// TIA Portal V15.1 export
// export: Created 2024-05-17T05:38:48.6670872Z, ExportSetting WithDefaults, DisplayName Totally Integrated Automation Portal, DisplayVersion V15.1 Update 5, DisplayName TIA Portal Openness, DisplayVersion V15.1 Update 5, DisplayName SINAMICS Startdrive Advanced, DisplayVersion V15.1, DisplayName G130, G150, S120, S150, SINAMICS MV, S210, DisplayVersion V15.1, DisplayName G110M, G120, G120C, G120D, G120P, DisplayVersion V15.1, DisplayName STEP 7 Professional, DisplayVersion V15.1 Update 5, DisplayName STEP 7 Safety, DisplayVersion V15.1, DisplayName WinCC Professional, DisplayVersion V15.1 Update 5, DisplayName SIMATIC Visualization Architect, DisplayVersion V15.1
FUNCTION_BLOCK "LGBLiftTable3Pos1S4Det-MoviFitFCPN"   // FB6652, FBD
TITLE = LGBLiftTable3Pos1S4Det-MoviFitFCPN
{ S7_Optimized_Access := 'TRUE' }
AUTHOR : VCC
FAMILY : Tooling
VERSION : 0.0.0.0
// =============================================================================
// This module will be used for a unit with 2 stop positions, 1 speed and controlled by a
// SEW MoviFit PN frequency converter.
// It will get commands from higher level, evaluate the status of the interlock
// and give a finished in return when the task is completed.
// ============================================================================
// stored: AutoNumber false, IsIECCheckEnabled false, IsRetainMemResEnabled false, MemoryReserve 100, SetENOAutomatically False, UDAEnableTagReadback false
   VAR_INPUT
      I_PosSet { ExternalAccessible := 'False'; ExternalVisible := 'False'; ExternalWritable := 'False'} : Bool;   // Position Set Detection 1
      I_PosSetCheck { ExternalAccessible := 'False'; ExternalVisible := 'False'; ExternalWritable := 'False'} : Bool;   // Position Set Detection 2
      I_PosMiddle { ExternalAccessible := 'False'; ExternalVisible := 'False'; ExternalWritable := 'False'} : Bool;   // Position Middle Detection
      I_PosRes { ExternalAccessible := 'False'; ExternalVisible := 'False'; ExternalWritable := 'False'} : Bool;   // Position Reset Detection 1
      I_PosResCheck { ExternalAccessible := 'False'; ExternalVisible := 'False'; ExternalWritable := 'False'} : Bool;   // Position Reset Detection 2
      I_SetBegin { ExternalAccessible := 'False'; ExternalVisible := 'False'; ExternalWritable := 'False'} : Bool;   // Function Set begin selection
      I_MiddleBegin { ExternalAccessible := 'False'; ExternalVisible := 'False'; ExternalWritable := 'False'} : Bool;   // Function Middle begin selection
      I_ResBegin { ExternalAccessible := 'False'; ExternalVisible := 'False'; ExternalWritable := 'False'} : Bool;   // Function Reset begin selection
      I_PBSet { ExternalAccessible := 'False'; ExternalVisible := 'False'; ExternalWritable := 'False'} : Bool;   // Push button for Set direction used in manual
      I_PBReset { ExternalAccessible := 'False'; ExternalVisible := 'False'; ExternalWritable := 'False'} : Bool;   // Push button for reset direcion used in manual
      I_SetIntlkOK { ExternalAccessible := 'False'; ExternalVisible := 'False'; ExternalWritable := 'False'} : Bool;   // Set Interlock
      I_ResIntlkOK { ExternalAccessible := 'False'; ExternalVisible := 'False'; ExternalWritable := 'False'} : Bool;   // Reset Interlock
      I_MotorProtection { ExternalAccessible := 'False'; ExternalVisible := 'False'; ExternalWritable := 'False'} : Bool;   // Motor protection
      I_ReleaseBrake { ExternalAccessible := 'False'; ExternalVisible := 'False'; ExternalWritable := 'False'} : Bool;   // Release brake
      I_SafetyOk { ExternalAccessible := 'False'; ExternalVisible := 'False'; ExternalWritable := 'False'} : Bool;   // Safety Ok
      I_MotionStopOk { ExternalAccessible := 'False'; ExternalVisible := 'False'; ExternalWritable := 'False'} : Bool;   // Safety Ok / The motion stop is Ok
      I_HighSpeed { ExternalAccessible := 'False'; ExternalVisible := 'False'; ExternalWritable := 'False'} : Real;   // High speed Value (set-up %)
      I_SafetyStatusWord { ExternalAccessible := 'False'; ExternalVisible := 'False'; ExternalWritable := 'False'} : Word;   // Safety Status
      I_SafetyControlWord { ExternalAccessible := 'False'; ExternalVisible := 'False'; ExternalWritable := 'False'} : Word;   // Safety Control Word
   END_VAR
   VAR_OUTPUT
      O_SetPos { ExternalAccessible := 'False'; ExternalVisible := 'False'; ExternalWritable := 'False'} : Bool;   // In Position Set
      O_MiddlePos { ExternalAccessible := 'False'; ExternalVisible := 'False'; ExternalWritable := 'False'} : Bool;   // In Position Middle
      O_ResPos { ExternalAccessible := 'False'; ExternalVisible := 'False'; ExternalWritable := 'False'} : Bool;   // In Position Reset
      O_ReleaseBrake { ExternalAccessible := 'False'; ExternalVisible := 'False'; ExternalWritable := 'False'} : Bool;   // Release the brake of the motor
      O_Active { ExternalAccessible := 'False'; ExternalVisible := 'False'; ExternalWritable := 'False'} : Bool;   // Motor Active
      O_FuncRunning { ExternalAccessible := 'False'; ExternalVisible := 'False'; ExternalWritable := 'False'} : Bool;   // Signal that the function is busy
      O_SetFinished { ExternalAccessible := 'False'; ExternalVisible := 'False'; ExternalWritable := 'False'} : Bool;   // Function Set finished to Master Sequencing
      O_MiddleFinished { ExternalAccessible := 'False'; ExternalVisible := 'False'; ExternalWritable := 'False'} : Bool;   // Function Middle finished to Master Sequencing
      O_ResFinished { ExternalAccessible := 'False'; ExternalVisible := 'False'; ExternalWritable := 'False'} : Bool;   // Function Reset finished to Master Sequencing
      O_LEDSet { ExternalAccessible := 'False'; ExternalVisible := 'False'; ExternalWritable := 'False'} : Bool;   // Ledindication / Led indication for Set
      O_LEDMiddle { ExternalAccessible := 'False'; ExternalVisible := 'False'; ExternalWritable := 'False'} : Bool;   // Ledindication / Led indication for Middle
      O_LEDRes { ExternalAccessible := 'False'; ExternalVisible := 'False'; ExternalWritable := 'False'} : Bool;   // Ledindication / Led indication for Reset
      O_ReadyForOperation { ExternalAccessible := 'False'; ExternalVisible := 'False'; ExternalWritable := 'False'} : Bool;   // Ready for operation
      O_AlarmABCondition { ExternalAccessible := 'False'; ExternalVisible := 'False'; ExternalWritable := 'False'} : Bool;   // Alarm AB condition
      O_AlarmA { ExternalAccessible := 'False'; ExternalVisible := 'False'; ExternalWritable := 'False'} : Bool;   // Alarm A
      O_AlarmB { ExternalAccessible := 'False'; ExternalVisible := 'False'; ExternalWritable := 'False'} : Bool;   // Alarm B
      O_AlarmC { ExternalAccessible := 'False'; ExternalVisible := 'False'; ExternalWritable := 'False'} : Bool;   // Alarm C
      O_AlarmD { ExternalAccessible := 'False'; ExternalVisible := 'False'; ExternalWritable := 'False'} : Bool;   // Alarm D
      H_AlarmDWord { ExternalAccessible := 'False'; ExternalVisible := 'False'; ExternalWritable := 'False'} : DWord;   // Alarm Word
      H_AlarmDWord2 { ExternalAccessible := 'False'; ExternalVisible := 'False'; ExternalWritable := 'False'} : DWord;   // Alarm Word
   END_VAR
   VAR_IN_OUT
      IO_Modes : "Modes";
      C_Config : "LiftTable3Pos1S4DetMoviFitFCPNConfig";
      H_HMI : "H_HMI";
      "H_GBLiftTable3Pos1S4Det-MoviFitFCPN" : "H_GBLiftTable3Pos1S4Det-MoviFitFCPN";
   END_VAR
   VAR
      _MovFunc3Pos { ExternalAccessible := 'False'; ExternalVisible := 'False'; ExternalWritable := 'False'} : "LMovFnc3Pos";   // FB
      _StopPos { ExternalAccessible := 'False'; ExternalVisible := 'False'; ExternalWritable := 'False'} : "L3StopPos";   // FB
      _Motor { ExternalAccessible := 'False'; ExternalVisible := 'False'; ExternalWritable := 'False'} : "LGBMotor2W2S-MoviFitFCPN";   // FB
      _SetDetMissing { ExternalAccessible := 'False'; ExternalVisible := 'False'; ExternalWritable := 'False'} : "LTimer";   // Timer
      _ResDetMissing { ExternalAccessible := 'False'; ExternalVisible := 'False'; ExternalWritable := 'False'} : "LTimer";   // Timer
      H_FncSelInHMI { ExternalAccessible := 'False'; ExternalVisible := 'False'; ExternalWritable := 'False'} : Bool;
      AA_MotorProtection { ExternalAccessible := 'False'; ExternalVisible := 'False'; ExternalWritable := 'False'} : Bool;   // Motorprotection Not Ok / Motor Protection Tripped
      AA_SafetySwitch { ExternalAccessible := 'False'; ExternalVisible := 'False'; ExternalWritable := 'False'} : Bool;   // Safety Switch Not Ok
      AB_STO { ExternalAccessible := 'False'; ExternalVisible := 'False'; ExternalWritable := 'False'} : Bool;   // Safety Switch Not Ok / Safety output to drive is active but no response from drive that the safety is ok
      AB_Alarm { ExternalAccessible := 'False'; ExternalVisible := 'False'; ExternalWritable := 'False'} : Bool;   // Frequency Control / Alarm Frequency Control
      AB_KeepPosSetAlm { ExternalAccessible := 'False'; ExternalVisible := 'False'; ExternalWritable := 'False'} : Bool;   // Position Supervision Set Position / Lost Set Position
      AB_KeepPosMiddleAlm { ExternalAccessible := 'False'; ExternalVisible := 'False'; ExternalWritable := 'False'} : Bool;   // Position Supervision Set Position / Lost Middle Position
      AB_KeepPosResAlm { ExternalAccessible := 'False'; ExternalVisible := 'False'; ExternalWritable := 'False'} : Bool;   // Position Supervision Reset Position / Lost Reset Position
      AB_OvtSetAlm { ExternalAccessible := 'False'; ExternalVisible := 'False'; ExternalWritable := 'False'} : Bool;   // Timeout Set / TimeOut Set Direction
      AB_OvtMiddleAlm { ExternalAccessible := 'False'; ExternalVisible := 'False'; ExternalWritable := 'False'} : Bool;   // Timeout Set / TimeOut Middle Direction
      AB_OvtResAlm { ExternalAccessible := 'False'; ExternalVisible := 'False'; ExternalWritable := 'False'} : Bool;   // Timeout Reset / TimeOut Reset Direction
      AB_MoreDetAlm { ExternalAccessible := 'False'; ExternalVisible := 'False'; ExternalWritable := 'False'} : Bool;   // More than One Detection On at the same Time
      AB_SetDet1Missing { ExternalAccessible := 'False'; ExternalVisible := 'False'; ExternalWritable := 'False'} : Bool;   // Set Detector Signal Missing
      AB_SetDet2Missing { ExternalAccessible := 'False'; ExternalVisible := 'False'; ExternalWritable := 'False'} : Bool;   // Set Check Detector Signal Missing
      AB_ResDet1Missing { ExternalAccessible := 'False'; ExternalVisible := 'False'; ExternalWritable := 'False'} : Bool;   // Reset Detector Signal Missing
      AB_ResDet2Missing { ExternalAccessible := 'False'; ExternalVisible := 'False'; ExternalWritable := 'False'} : Bool;   // Reset Check Detector Signal Missing
      AC_KeepPosSetAlm { ExternalAccessible := 'False'; ExternalVisible := 'False'; ExternalWritable := 'False'} : Bool;   // Lost Set Position
      AC_KeepPosMiddleAlm { ExternalAccessible := 'False'; ExternalVisible := 'False'; ExternalWritable := 'False'} : Bool;   // Lost Set Position / Lost Middle Position
      AC_KeepPosResAlm { ExternalAccessible := 'False'; ExternalVisible := 'False'; ExternalWritable := 'False'} : Bool;   // Lost Reset Position
      AC_OvtSetAlm { ExternalAccessible := 'False'; ExternalVisible := 'False'; ExternalWritable := 'False'} : Bool;   // Timeout Set / TimeOut Set Direction
      AC_OvtMiddleAlm { ExternalAccessible := 'False'; ExternalVisible := 'False'; ExternalWritable := 'False'} : Bool;   // Timeout Set / TimeOut Middle Direction
      AC_OvtResAlm { ExternalAccessible := 'False'; ExternalVisible := 'False'; ExternalWritable := 'False'} : Bool;   // Timeout Reset / TimeOut Reset Direction
      AC_MoreDetAlm { ExternalAccessible := 'False'; ExternalVisible := 'False'; ExternalWritable := 'False'} : Bool;   // More than One Detection On at the same Time
      AC_SetDet1Missing { ExternalAccessible := 'False'; ExternalVisible := 'False'; ExternalWritable := 'False'} : Bool;   // Set Detector Signal Missing
      AC_SetDet2Missing { ExternalAccessible := 'False'; ExternalVisible := 'False'; ExternalWritable := 'False'} : Bool;   // Set Check Detector Signal Missing
      AC_ResDet1Missing { ExternalAccessible := 'False'; ExternalVisible := 'False'; ExternalWritable := 'False'} : Bool;   // Reset Detector Signal Missing
      AC_ResDet2Missing { ExternalAccessible := 'False'; ExternalVisible := 'False'; ExternalWritable := 'False'} : Bool;   // Reset Check Detector Signal Missing
      AD_OvtSetWarn { ExternalAccessible := 'False'; ExternalVisible := 'False'; ExternalWritable := 'False'} : Bool;   // Timeout Set / TimeOut Set Direction
      AD_OvtMiddleWarn { ExternalAccessible := 'False'; ExternalVisible := 'False'; ExternalWritable := 'False'} : Bool;   // TimeOut To Middle / Timeout Middle
      AD_OvtResWarn { ExternalAccessible := 'False'; ExternalVisible := 'False'; ExternalWritable := 'False'} : Bool;   // Timeout Reset / TimeOut Reset Direction
      AD_IntlkSetAlm { ExternalAccessible := 'False'; ExternalVisible := 'False'; ExternalWritable := 'False'} : Bool;   // Interlock Set
      AD_IntlkMiddleAlm { ExternalAccessible := 'False'; ExternalVisible := 'False'; ExternalWritable := 'False'} : Bool;   // Interlock Middle
      AD_IntlkResAlm { ExternalAccessible := 'False'; ExternalVisible := 'False'; ExternalWritable := 'False'} : Bool;   // Interlock Reset
      AD_Warning { ExternalAccessible := 'False'; ExternalVisible := 'False'; ExternalWritable := 'False'} : Bool;   // Frequency Control / Warning Frequency Control
      AA_NoBusControl { ExternalAccessible := 'False'; ExternalVisible := 'False'; ExternalWritable := 'False'} : Bool;   // Bus control inactive / Bus Control Inactive Frequency Control
      AD_MotionStop { ExternalAccessible := 'False'; ExternalVisible := 'False'; ExternalWritable := 'False'} : Bool;   // Motion Stop
      AC_ConfigCalibrationAlm { ExternalAccessible := 'False'; ExternalVisible := 'False'; ExternalWritable := 'False'} : Bool;   // The Config values for Warming/Alarm time must be ALL zero or ALL different from zero
      AD_CalibrationWarn { ExternalAccessible := 'False'; ExternalVisible := 'False'; ExternalWritable := 'False'} : Bool;   // No High speed selected so Calibration is not possible
      AC_ConfigRampAlm { ExternalAccessible := 'False'; ExternalVisible := 'False'; ExternalWritable := 'False'} : Bool;   // The config value for the ramp is not correct, must be zero or the config values for the calculation of the ramp must be ALL zero
      AC_ConfigRampCalcAlm { ExternalAccessible := 'False'; ExternalVisible := 'False'; ExternalWritable := 'False'} : Bool;   // The config values for the calculation of the ramp must be ALL different from zero
      PODataNotEnabled { ExternalAccessible := 'False'; ExternalVisible := 'False'; ExternalWritable := 'False'} : Bool;   // Bus control inactive
      SafetyOk { ExternalAccessible := 'False'; ExternalVisible := 'False'; ExternalWritable := 'False'} : Bool;   // Safety Ok
      SetPos { ExternalAccessible := 'False'; ExternalVisible := 'False'; ExternalWritable := 'False'} : Bool;   // Set position
      MiddlePos { ExternalAccessible := 'False'; ExternalVisible := 'False'; ExternalWritable := 'False'} : Bool;   // Middle Position
      ResPos { ExternalAccessible := 'False'; ExternalVisible := 'False'; ExternalWritable := 'False'} : Bool;   // Reset position
      AlarmA { ExternalAccessible := 'False'; ExternalVisible := 'False'; ExternalWritable := 'False'} : Bool;   // Alarm A
      AlarmB { ExternalAccessible := 'False'; ExternalVisible := 'False'; ExternalWritable := 'False'} : Bool;   // Alarm B
      AlarmC { ExternalAccessible := 'False'; ExternalVisible := 'False'; ExternalWritable := 'False'} : Bool;   // Alarm C
      AlarmD { ExternalAccessible := 'False'; ExternalVisible := 'False'; ExternalWritable := 'False'} : Bool;   // Alarm D
      SetIntlkOK { ExternalAccessible := 'False'; ExternalVisible := 'False'; ExternalWritable := 'False'} : Bool;   // Set Interlock
      MiddleIntlkOK { ExternalAccessible := 'False'; ExternalVisible := 'False'; ExternalWritable := 'False'} : Bool;   // Set Interlock / Middle Interlock
      ResIntlkOK { ExternalAccessible := 'False'; ExternalVisible := 'False'; ExternalWritable := 'False'} : Bool;   // Reset Interlock
      FuncRunning { ExternalAccessible := 'False'; ExternalVisible := 'False'; ExternalWritable := 'False'} : Bool;   // Function running
      MovFuncAlmCond { ExternalAccessible := 'False'; ExternalVisible := 'False'; ExternalWritable := 'False'} : Bool;   // Move function Alarm Condition
      StopPosAlmCond { ExternalAccessible := 'False'; ExternalVisible := 'False'; ExternalWritable := 'False'} : Bool;   // Stop posistion Alarm Condition
      KeepPosSetAlm { ExternalAccessible := 'False'; ExternalVisible := 'False'; ExternalWritable := 'False'} : Bool;   // Alarm Keep Position Set Position
      KeepPosMiddleAlm { ExternalAccessible := 'False'; ExternalVisible := 'False'; ExternalWritable := 'False'} : Bool;   // Keep Position Middle Alarm
      KeepPosResAlm { ExternalAccessible := 'False'; ExternalVisible := 'False'; ExternalWritable := 'False'} : Bool;   // Position Supervision Reset Position
      OvtSetAlm { ExternalAccessible := 'False'; ExternalVisible := 'False'; ExternalWritable := 'False'} : Bool;   // Timeout Set
      OvtMiddleAlm { ExternalAccessible := 'False'; ExternalVisible := 'False'; ExternalWritable := 'False'} : Bool;   // Overtime goto Middle Alarm
      OvtResAlm { ExternalAccessible := 'False'; ExternalVisible := 'False'; ExternalWritable := 'False'} : Bool;   // Overtime reset Alarm
      OneSetDetMissing { ExternalAccessible := 'False'; ExternalVisible := 'False'; ExternalWritable := 'False'} : Bool;   // One Set detector is missing
      OneResDetMissing { ExternalAccessible := 'False'; ExternalVisible := 'False'; ExternalWritable := 'False'} : Bool;   // One Reset detector is missing
      DetectorMissing { ExternalAccessible := 'False'; ExternalVisible := 'False'; ExternalWritable := 'False'} : Bool;   // One detector is missing
      OutOfUse { ExternalAccessible := 'False'; ExternalVisible := 'False'; ExternalWritable := 'False'} : Bool;   // Out of use
      MotorLoopAlarmCond { ExternalAccessible := 'False'; ExternalVisible := 'False'; ExternalWritable := 'False'} : Bool;   // Motor loop Alarm Condition
      ReadyForOperation { ExternalAccessible := 'False'; ExternalVisible := 'False'; ExternalWritable := 'False'} : Bool;   // Motor Loop Ready for operation
      MotorLoopActive { ExternalAccessible := 'False'; ExternalVisible := 'False'; ExternalWritable := 'False'} : Bool;   // Motor Loop Active
      AlarmABCondition { ExternalAccessible := 'False'; ExternalVisible := 'False'; ExternalWritable := 'False'} : Bool;   // Alarm AB Condition
      ReleaseBrake { ExternalAccessible := 'False'; ExternalVisible := 'False'; ExternalWritable := 'False'} : Bool;   // Release brake
      MotorCmdSet { ExternalAccessible := 'False'; ExternalVisible := 'False'; ExternalWritable := 'False'} : Bool;   // Command to motorloop set
      MotorCmdRes { ExternalAccessible := 'False'; ExternalVisible := 'False'; ExternalWritable := 'False'} : Bool;   // Command to motorloop reset
      SetPosDelayd { ExternalAccessible := 'False'; ExternalVisible := 'False'; ExternalWritable := 'False'} : Bool;   // Set Position Delayed
      MiddlePosDelayd { ExternalAccessible := 'False'; ExternalVisible := 'False'; ExternalWritable := 'False'} : Bool;   // Middle Position Delayed
      ResPosDelayd { ExternalAccessible := 'False'; ExternalVisible := 'False'; ExternalWritable := 'False'} : Bool;   // Reset Position Delayed
   END_VAR
   VAR RETAIN
      MemPrevPosRes { ExternalAccessible := 'False'; ExternalVisible := 'False'; ExternalWritable := 'False'} : Bool;   // Memory previous position was Reset
   END_VAR
   VAR
      MoreThenOneDetAlm { ExternalAccessible := 'False'; ExternalVisible := 'False'; ExternalWritable := 'False'} : Bool;   // More then one detection Alarm
      CmdSet { ExternalAccessible := 'False'; ExternalVisible := 'False'; ExternalWritable := 'False'} : Bool;   // Command Set
      CmdMiddle { ExternalAccessible := 'False'; ExternalVisible := 'False'; ExternalWritable := 'False'} : Bool;   // Command Middle
      CmdRes { ExternalAccessible := 'False'; ExternalVisible := 'False'; ExternalWritable := 'False'} : Bool;   // Command Reset
      MiddleStartMan { ExternalAccessible := 'False'; ExternalVisible := 'False'; ExternalWritable := 'False'} : Bool;   // Middle pos reached
      MiddleReachedMan { ExternalAccessible := 'False'; ExternalVisible := 'False'; ExternalWritable := 'False'} : Bool;   // Middle pos reached
      MiddleReachedManSTOP { ExternalAccessible := 'False'; ExternalVisible := 'False'; ExternalWritable := 'False'} : Bool;   // Middle pos reached
      PosSetDelayTimer { ExternalAccessible := 'False'; ExternalVisible := 'False'; ExternalWritable := 'False'} : "LTimer";   // FB
      PosMiddleDelayTimer { ExternalAccessible := 'False'; ExternalVisible := 'False'; ExternalWritable := 'False'} : "LTimer";   // FB
      PosResDelayTimer { ExternalAccessible := 'False'; ExternalVisible := 'False'; ExternalWritable := 'False'} : "LTimer";   // FB
   END_VAR
   VAR_TEMP
      H_HMITemp : "H_HMI";   // Animation
      H_HMIMotor : "H_HMI";   // Temp
      TempDInt : DInt;   // Temp DInt
      RunTimeMaxMiddleWarn : DInt;   // Time in ms for overtime warning
      RunTimeMaxMiddleAlm : DInt;   // Time in ms for overtime alarm
   END_VAR
   VAR_TEMP   // added for the SCL form of the ladder/FBD networks
      _w1 : Bool;
   END_VAR
BEGIN

REGION Network 1: **** 1 - Inputs **** Set Position Delay Timer
   // Set Position Delay Timer
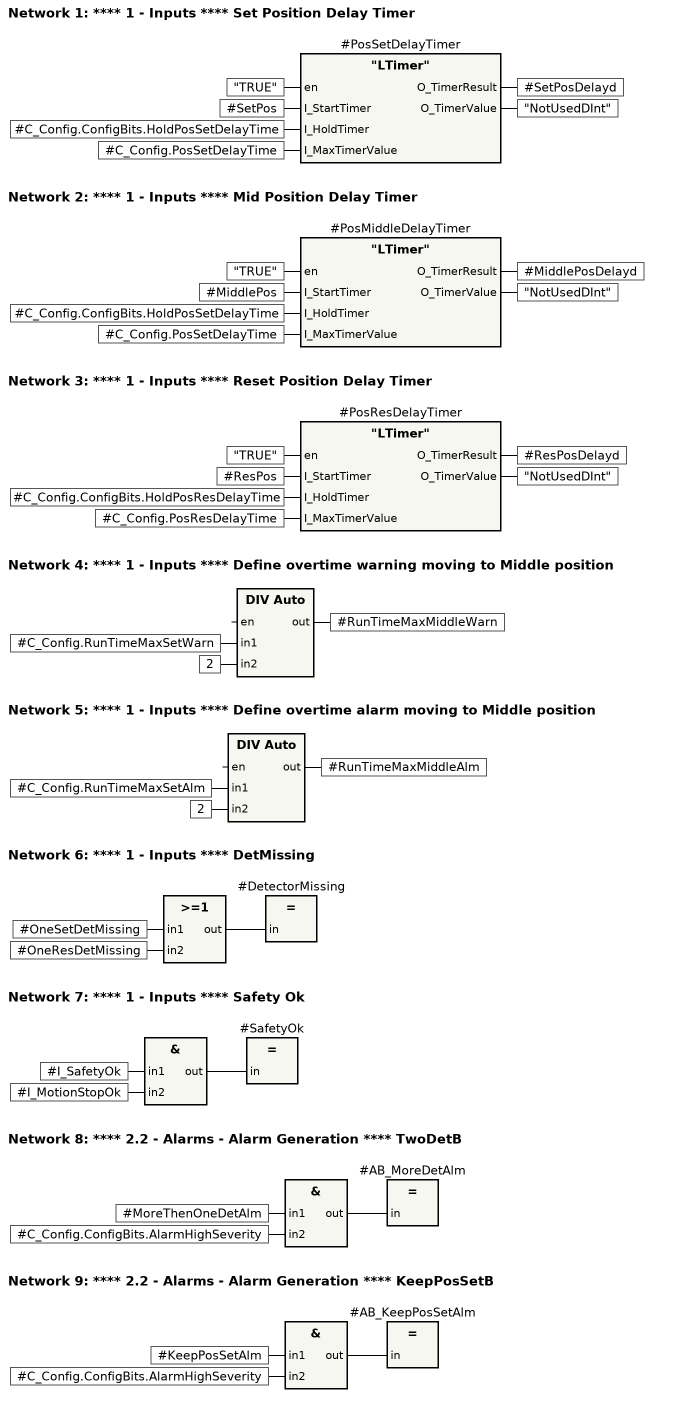
   IF "TRUE" THEN
       #PosSetDelayTimer(I_StartTimer := #SetPos,   // "LTimer"
                         I_HoldTimer := #C_Config.ConfigBits.HoldPosSetDelayTime,
                         I_MaxTimerValue := #C_Config.PosSetDelayTime,
                         O_TimerResult => #SetPosDelayd,
                         O_TimerValue => "NotUsedDInt");
   END_IF;
END_REGION

REGION Network 2: **** 1 - Inputs **** Mid Position Delay Timer
   // Middle Position Delay Timer
   IF "TRUE" THEN
       #PosMiddleDelayTimer(I_StartTimer := #MiddlePos,   // "LTimer"
                            I_HoldTimer := #C_Config.ConfigBits.HoldPosSetDelayTime,
                            I_MaxTimerValue := #C_Config.PosSetDelayTime,
                            O_TimerResult => #MiddlePosDelayd,
                            O_TimerValue => "NotUsedDInt");
   END_IF;
END_REGION

REGION Network 3: **** 1 - Inputs **** Reset Position Delay Timer
   // Reset Position Delay Timer
   IF "TRUE" THEN
       #PosResDelayTimer(I_StartTimer := #ResPos,   // "LTimer"
                         I_HoldTimer := #C_Config.ConfigBits.HoldPosResDelayTime,
                         I_MaxTimerValue := #C_Config.PosResDelayTime,
                         O_TimerResult => #ResPosDelayd,
                         O_TimerValue => "NotUsedDInt");
   END_IF;
END_REGION

REGION Network 4: **** 1 - Inputs **** Define overtime warning moving to Middle position
   // Define overtime warning moving to Middle position
   #RunTimeMaxMiddleWarn := #C_Config.RunTimeMaxSetWarn / 2;
END_REGION

REGION Network 5: **** 1 - Inputs **** Define overtime alarm moving to Middle position
   // Define overtime alarm moving to Middle position
   #RunTimeMaxMiddleAlm := #C_Config.RunTimeMaxSetAlm / 2;
END_REGION

REGION Network 6: **** 1 - Inputs **** DetMissing
   // Disable other Alarms when a detector is missing
   #DetectorMissing := #OneSetDetMissing OR #OneResDetMissing;
END_REGION

REGION Network 7: **** 1 - Inputs **** Safety Ok
   #SafetyOk := #I_SafetyOk AND #I_MotionStopOk;
END_REGION

REGION Network 8: **** 2.2 - Alarms - Alarm Generation **** TwoDetB
   // Two Detection B Alarm
   #AB_MoreDetAlm := #MoreThenOneDetAlm AND #C_Config.ConfigBits.AlarmHighSeverity;
END_REGION

REGION Network 9: **** 2.2 - Alarms - Alarm Generation **** KeepPosSetB
   // Keep position Set B Alarm
   #AB_KeepPosSetAlm := #KeepPosSetAlm AND #C_Config.ConfigBits.AlarmHighSeverity;
END_REGION

REGION Network 10: **** 2.2 - Alarms - Alarm Generation **** KeepPosSetB / **** 2.2 - Alarms - Alarm Generation **** KeepPosMiddleB
   // Keep position Set B Alarm / Keep position Middle B Alarm
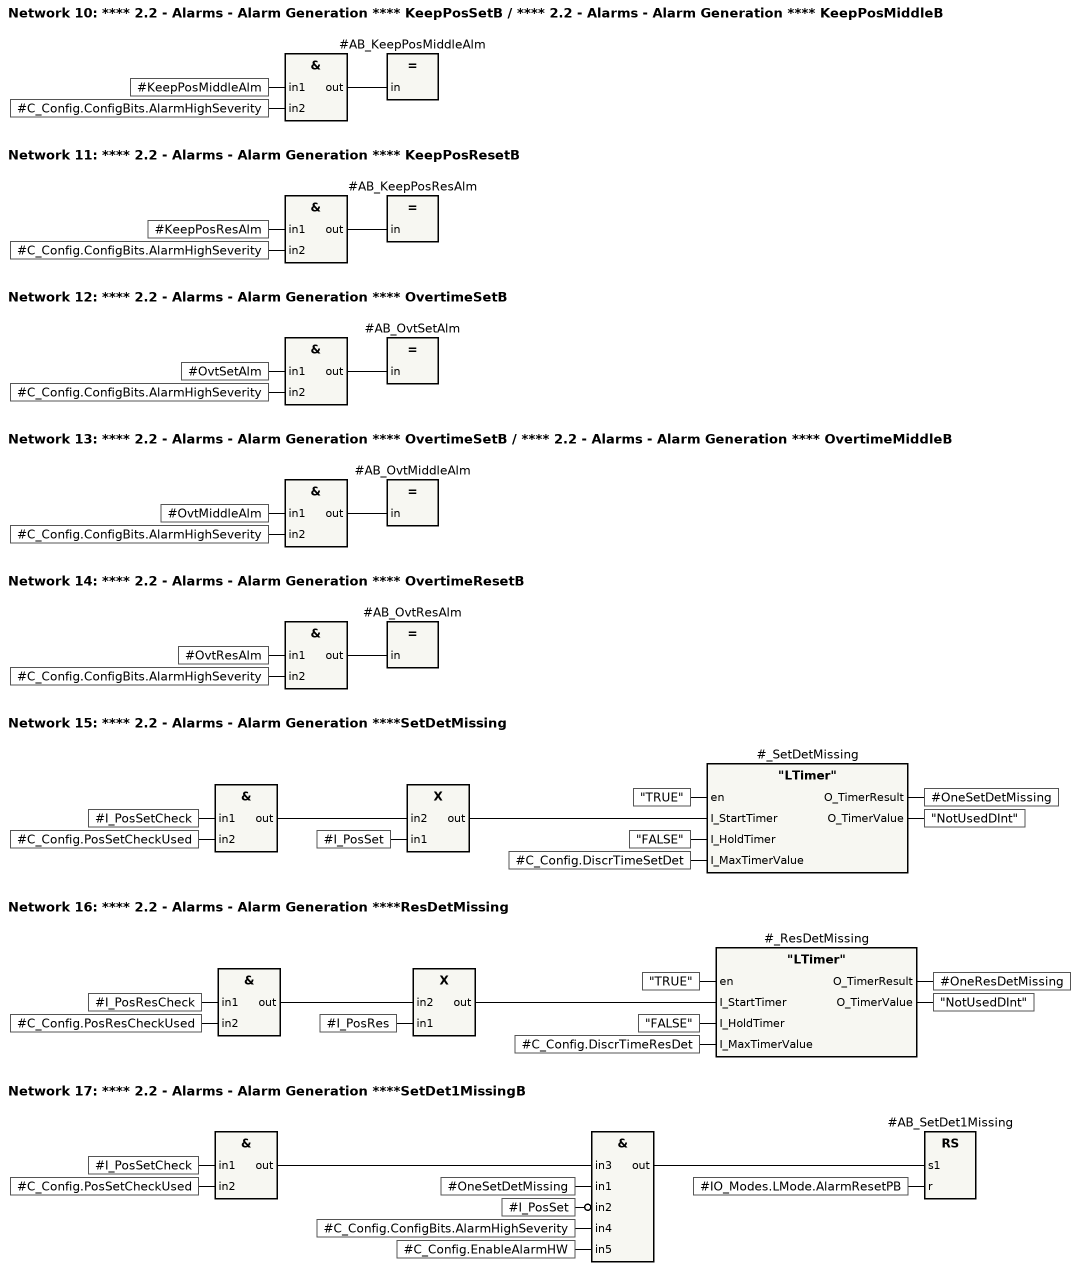
   #AB_KeepPosMiddleAlm := #KeepPosMiddleAlm AND #C_Config.ConfigBits.AlarmHighSeverity;
END_REGION

REGION Network 11: **** 2.2 - Alarms - Alarm Generation **** KeepPosResetB
   // Keep position reset B Alarm
   #AB_KeepPosResAlm := #KeepPosResAlm AND #C_Config.ConfigBits.AlarmHighSeverity;
END_REGION

REGION Network 12: **** 2.2 - Alarms - Alarm Generation **** OvertimeSetB
   // Overtime set B Alarm
   #AB_OvtSetAlm := #OvtSetAlm AND #C_Config.ConfigBits.AlarmHighSeverity;
END_REGION

REGION Network 13: **** 2.2 - Alarms - Alarm Generation **** OvertimeSetB / **** 2.2 - Alarms - Alarm Generation **** OvertimeMiddleB
   // Overtime set B Alarm / Overtime Middle B Alarm
   #AB_OvtMiddleAlm := #OvtMiddleAlm AND #C_Config.ConfigBits.AlarmHighSeverity;
END_REGION

REGION Network 14: **** 2.2 - Alarms - Alarm Generation **** OvertimeResetB
   // Overtime reset B Alarm
   #AB_OvtResAlm := #OvtResAlm AND #C_Config.ConfigBits.AlarmHighSeverity;
END_REGION

REGION Network 15: **** 2.2 - Alarms - Alarm Generation ****SetDetMissing
   // Any Set detector missing
   IF "TRUE" THEN
       #_SetDetMissing(I_StartTimer := (#I_PosSetCheck AND #C_Config.PosSetCheckUsed) XOR #I_PosSet,   // "LTimer"
                       I_HoldTimer := "FALSE",
                       I_MaxTimerValue := #C_Config.DiscrTimeSetDet,
                       O_TimerResult => #OneSetDetMissing,
                       O_TimerValue => "NotUsedDInt");
   END_IF;
END_REGION

REGION Network 16: **** 2.2 - Alarms - Alarm Generation ****ResDetMissing
   // Any Reset detector missing
   IF "TRUE" THEN
       #_ResDetMissing(I_StartTimer := (#I_PosResCheck AND #C_Config.PosResCheckUsed) XOR #I_PosRes,   // "LTimer"
                       I_HoldTimer := "FALSE",
                       I_MaxTimerValue := #C_Config.DiscrTimeResDet,
                       O_TimerResult => #OneResDetMissing,
                       O_TimerValue => "NotUsedDInt");
   END_IF;
END_REGION

REGION Network 17: **** 2.2 - Alarms - Alarm Generation ****SetDet1MissingB
   // Set detector 1 missing
   IF #IO_Modes.LMode.AlarmResetPB THEN
       #AB_SetDet1Missing := FALSE;   // RS flip-flop
   END_IF;
   IF #I_PosSetCheck AND #C_Config.PosSetCheckUsed AND #OneSetDetMissing AND NOT #I_PosSet AND #C_Config.ConfigBits.AlarmHighSeverity AND #C_Config.EnableAlarmHW THEN
       #AB_SetDet1Missing := TRUE;
   END_IF;
END_REGION

REGION Network 18: **** 2.2 - Alarms - Alarm Generation ****SetDet2MissingB
   // Set detector 2 missing
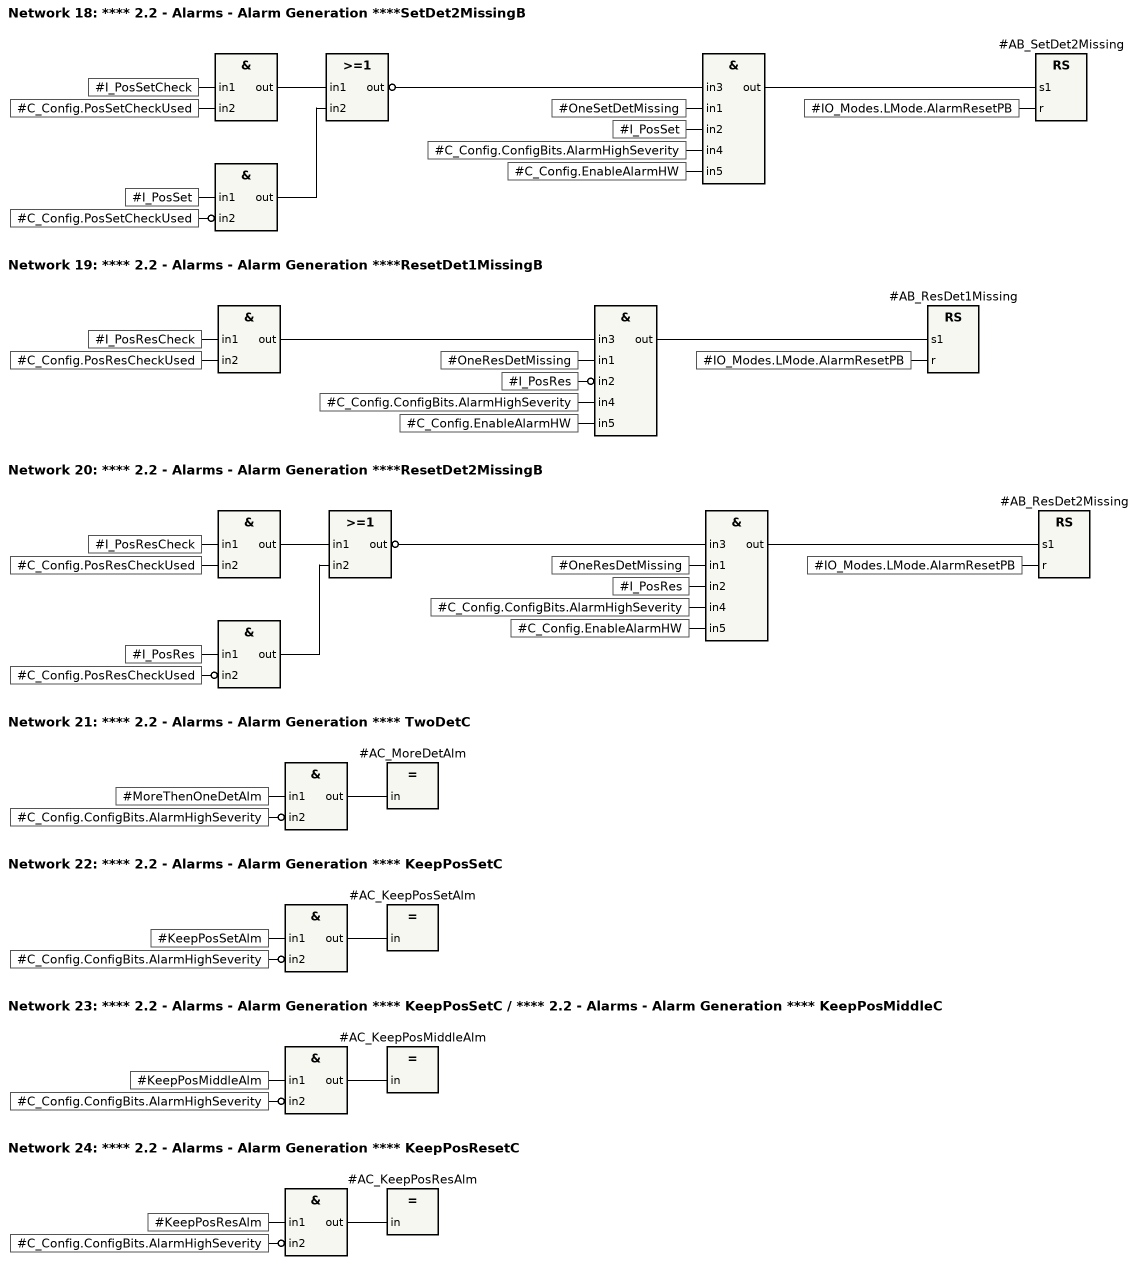
   IF #IO_Modes.LMode.AlarmResetPB THEN
       #AB_SetDet2Missing := FALSE;   // RS flip-flop
   END_IF;
   IF NOT ((#I_PosSetCheck AND #C_Config.PosSetCheckUsed) OR (#I_PosSet AND NOT #C_Config.PosSetCheckUsed)) AND #OneSetDetMissing AND #I_PosSet AND #C_Config.ConfigBits.AlarmHighSeverity AND #C_Config.EnableAlarmHW THEN
       #AB_SetDet2Missing := TRUE;
   END_IF;
END_REGION

REGION Network 19: **** 2.2 - Alarms - Alarm Generation ****ResetDet1MissingB
   // Reset detector 1 missing
   IF #IO_Modes.LMode.AlarmResetPB THEN
       #AB_ResDet1Missing := FALSE;   // RS flip-flop
   END_IF;
   IF #I_PosResCheck AND #C_Config.PosResCheckUsed AND #OneResDetMissing AND NOT #I_PosRes AND #C_Config.ConfigBits.AlarmHighSeverity AND #C_Config.EnableAlarmHW THEN
       #AB_ResDet1Missing := TRUE;
   END_IF;
END_REGION

REGION Network 20: **** 2.2 - Alarms - Alarm Generation ****ResetDet2MissingB
   // Reset detector 2 missing
   IF #IO_Modes.LMode.AlarmResetPB THEN
       #AB_ResDet2Missing := FALSE;   // RS flip-flop
   END_IF;
   IF NOT ((#I_PosResCheck AND #C_Config.PosResCheckUsed) OR (#I_PosRes AND NOT #C_Config.PosResCheckUsed)) AND #OneResDetMissing AND #I_PosRes AND #C_Config.ConfigBits.AlarmHighSeverity AND #C_Config.EnableAlarmHW THEN
       #AB_ResDet2Missing := TRUE;
   END_IF;
END_REGION

REGION Network 21: **** 2.2 - Alarms - Alarm Generation **** TwoDetC
   // Two Detection C Alarm
   #AC_MoreDetAlm := #MoreThenOneDetAlm AND NOT #C_Config.ConfigBits.AlarmHighSeverity;
END_REGION

REGION Network 22: **** 2.2 - Alarms - Alarm Generation **** KeepPosSetC
   // Keep position Set C Alarm
   #AC_KeepPosSetAlm := #KeepPosSetAlm AND NOT #C_Config.ConfigBits.AlarmHighSeverity;
END_REGION

REGION Network 23: **** 2.2 - Alarms - Alarm Generation **** KeepPosSetC / **** 2.2 - Alarms - Alarm Generation **** KeepPosMiddleC
   // Keep position Set C Alarm / Keep position Middle C Alarm
   #AC_KeepPosMiddleAlm := #KeepPosMiddleAlm AND NOT #C_Config.ConfigBits.AlarmHighSeverity;
END_REGION

REGION Network 24: **** 2.2 - Alarms - Alarm Generation **** KeepPosResetC
   // Keep position reset C Alarm
   #AC_KeepPosResAlm := #KeepPosResAlm AND NOT #C_Config.ConfigBits.AlarmHighSeverity;
END_REGION

REGION Network 25: **** 2.2 - Alarms - Alarm Generation **** OvertimeSetC
   // Overtime set C Alarm
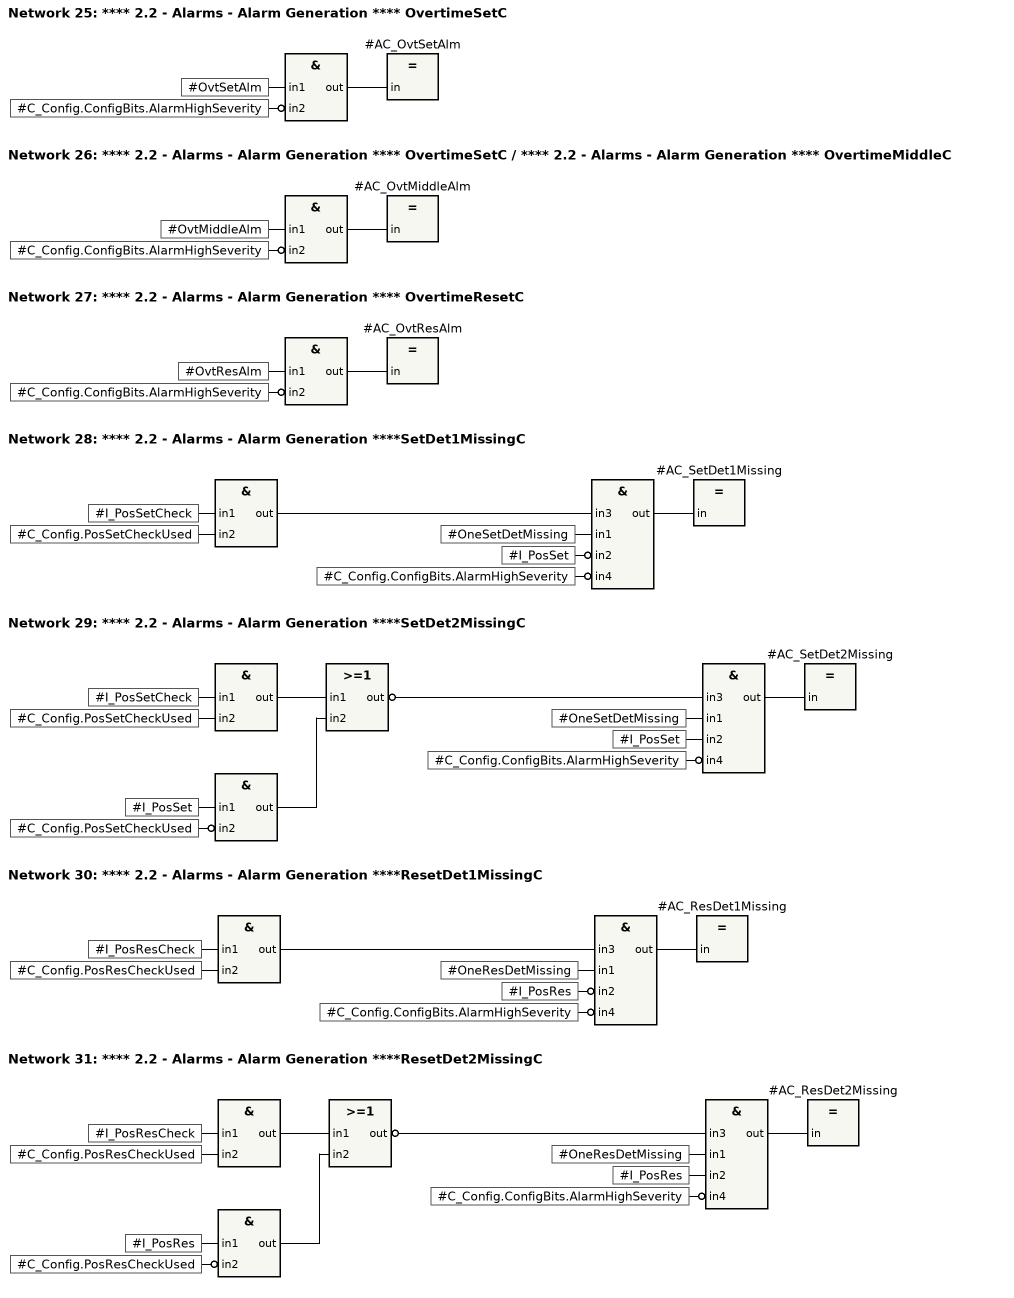
   #AC_OvtSetAlm := #OvtSetAlm AND NOT #C_Config.ConfigBits.AlarmHighSeverity;
END_REGION

REGION Network 26: **** 2.2 - Alarms - Alarm Generation **** OvertimeSetC / **** 2.2 - Alarms - Alarm Generation **** OvertimeMiddleC
   // Overtime set C Alarm / Overtime Middle C Alarm
   #AC_OvtMiddleAlm := #OvtMiddleAlm AND NOT #C_Config.ConfigBits.AlarmHighSeverity;
END_REGION

REGION Network 27: **** 2.2 - Alarms - Alarm Generation **** OvertimeResetC
   // Overtime reset C Alarm
   #AC_OvtResAlm := #OvtResAlm AND NOT #C_Config.ConfigBits.AlarmHighSeverity;
END_REGION

REGION Network 28: **** 2.2 - Alarms - Alarm Generation ****SetDet1MissingC
   // Set detector 1 missing
   #AC_SetDet1Missing := #I_PosSetCheck AND #C_Config.PosSetCheckUsed AND #OneSetDetMissing AND NOT #I_PosSet AND NOT #C_Config.ConfigBits.AlarmHighSeverity;
END_REGION

REGION Network 29: **** 2.2 - Alarms - Alarm Generation ****SetDet2MissingC
   // Set detector 2 missing
   #AC_SetDet2Missing := NOT ((#I_PosSetCheck AND #C_Config.PosSetCheckUsed) OR (#I_PosSet AND NOT #C_Config.PosSetCheckUsed)) AND #OneSetDetMissing AND #I_PosSet AND NOT #C_Config.ConfigBits.AlarmHighSeverity;
END_REGION

REGION Network 30: **** 2.2 - Alarms - Alarm Generation ****ResetDet1MissingC
   // Reset detector 1 missing
   #AC_ResDet1Missing := #I_PosResCheck AND #C_Config.PosResCheckUsed AND #OneResDetMissing AND NOT #I_PosRes AND NOT #C_Config.ConfigBits.AlarmHighSeverity;
END_REGION

REGION Network 31: **** 2.2 - Alarms - Alarm Generation ****ResetDet2MissingC
   // Reset detector 2 missing
   #AC_ResDet2Missing := NOT ((#I_PosResCheck AND #C_Config.PosResCheckUsed) OR (#I_PosRes AND NOT #C_Config.PosResCheckUsed)) AND #OneResDetMissing AND #I_PosRes AND NOT #C_Config.ConfigBits.AlarmHighSeverity;
END_REGION

REGION Network 32: **** 2.2 - Alarms - Alarm Generation **** No bus control
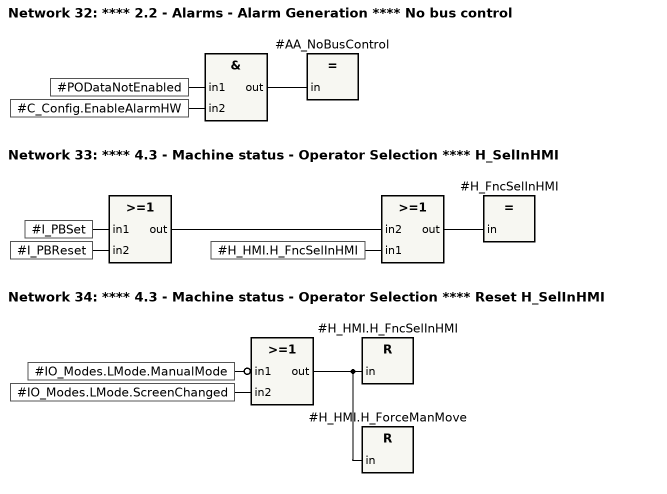
   #AA_NoBusControl := #PODataNotEnabled AND #C_Config.EnableAlarmHW;
END_REGION

REGION Network 33: **** 4.3 - Machine status - Operator Selection **** H_SelInHMI
   #H_FncSelInHMI := #I_PBSet OR #I_PBReset OR #H_HMI.H_FncSelInHMI;
END_REGION

REGION Network 34: **** 4.3 - Machine status - Operator Selection **** Reset H_SelInHMI
   // Reset H_SelInHMI
   IF NOT #IO_Modes.LMode.ManualMode OR #IO_Modes.LMode.ScreenChanged THEN
       #H_HMI.H_FncSelInHMI := FALSE;
       #H_HMI.H_ForceManMove := FALSE;
   END_IF;
END_REGION

REGION Network 35: **** 4.6 - Machine status - Indication **** Icon Animation
   // Icon animation
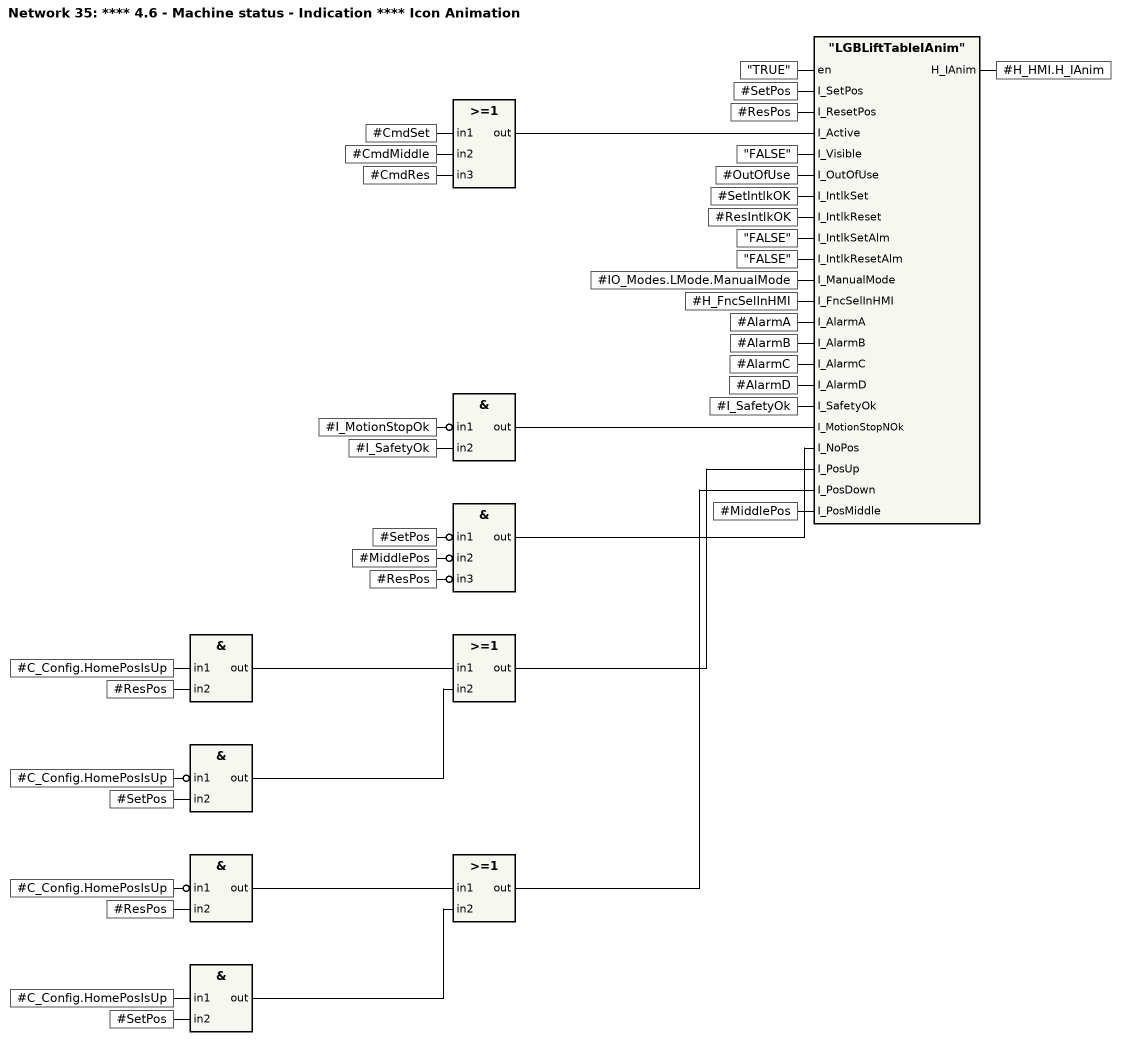
   IF "TRUE" THEN
       "LGBLiftTableIAnim"(I_SetPos := #SetPos,
                           I_ResetPos := #ResPos,
                           I_Active := #CmdSet OR #CmdMiddle OR #CmdRes,
                           I_Visible := "FALSE",
                           I_OutOfUse := #OutOfUse,
                           I_IntlkSet := #SetIntlkOK,
                           I_IntlkReset := #ResIntlkOK,
                           I_IntlkSetAlm := "FALSE",
                           I_IntlkResetAlm := "FALSE",
                           I_ManualMode := #IO_Modes.LMode.ManualMode,
                           I_FncSelInHMI := #H_FncSelInHMI,
                           I_AlarmA := #AlarmA,
                           I_AlarmB := #AlarmB,
                           I_AlarmC := #AlarmC,
                           I_AlarmD := #AlarmD,
                           I_SafetyOk := #I_SafetyOk,
                           I_MotionStopNOk := NOT #I_MotionStopOk AND #I_SafetyOk,
                           I_NoPos := NOT #SetPos AND NOT #MiddlePos AND NOT #ResPos,
                           I_PosUp := (#C_Config.HomePosIsUp AND #ResPos) OR (NOT #C_Config.HomePosIsUp AND #SetPos),
                           I_PosDown := (NOT #C_Config.HomePosIsUp AND #ResPos) OR (#C_Config.HomePosIsUp AND #SetPos),
                           I_PosMiddle := #MiddlePos,
                           H_IAnim => #H_HMI.H_IAnim);
   END_IF;
END_REGION

REGION Network 36: **** 4.6 - Machine status - Indication **** PosSetIAnim
   // Icon animation
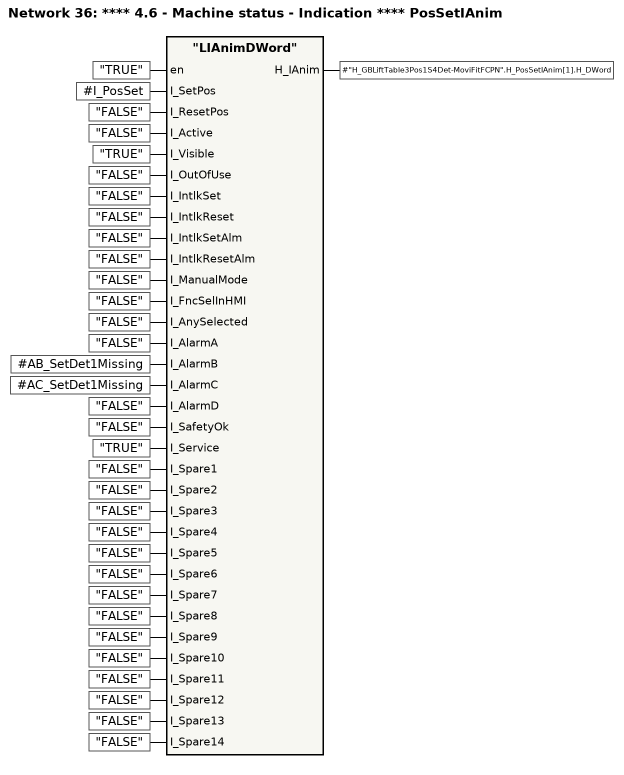
   IF "TRUE" THEN
       "LIAnimDWord"(I_SetPos := #I_PosSet,
                     I_ResetPos := "FALSE",
                     I_Active := "FALSE",
                     I_Visible := "TRUE",
                     I_OutOfUse := "FALSE",
                     I_IntlkSet := "FALSE",
                     I_IntlkReset := "FALSE",
                     I_IntlkSetAlm := "FALSE",
                     I_IntlkResetAlm := "FALSE",
                     I_ManualMode := "FALSE",
                     I_FncSelInHMI := "FALSE",
                     I_AnySelected := "FALSE",
                     I_AlarmA := "FALSE",
                     I_AlarmB := #AB_SetDet1Missing,
                     I_AlarmC := #AC_SetDet1Missing,
                     I_AlarmD := "FALSE",
                     I_SafetyOk := "FALSE",
                     I_Service := "TRUE",
                     I_Spare1 := "FALSE",
                     I_Spare2 := "FALSE",
                     I_Spare3 := "FALSE",
                     I_Spare4 := "FALSE",
                     I_Spare5 := "FALSE",
                     I_Spare6 := "FALSE",
                     I_Spare7 := "FALSE",
                     I_Spare8 := "FALSE",
                     I_Spare9 := "FALSE",
                     I_Spare10 := "FALSE",
                     I_Spare11 := "FALSE",
                     I_Spare12 := "FALSE",
                     I_Spare13 := "FALSE",
                     I_Spare14 := "FALSE",
                     H_IAnim => #"H_GBLiftTable3Pos1S4Det-MoviFitFCPN".H_PosSetIAnim[1].H_DWord);
   END_IF;
END_REGION

REGION Network 37: **** 4.6 - Machine status - Indication **** PosSetCheckIAnim
   // Icon animation
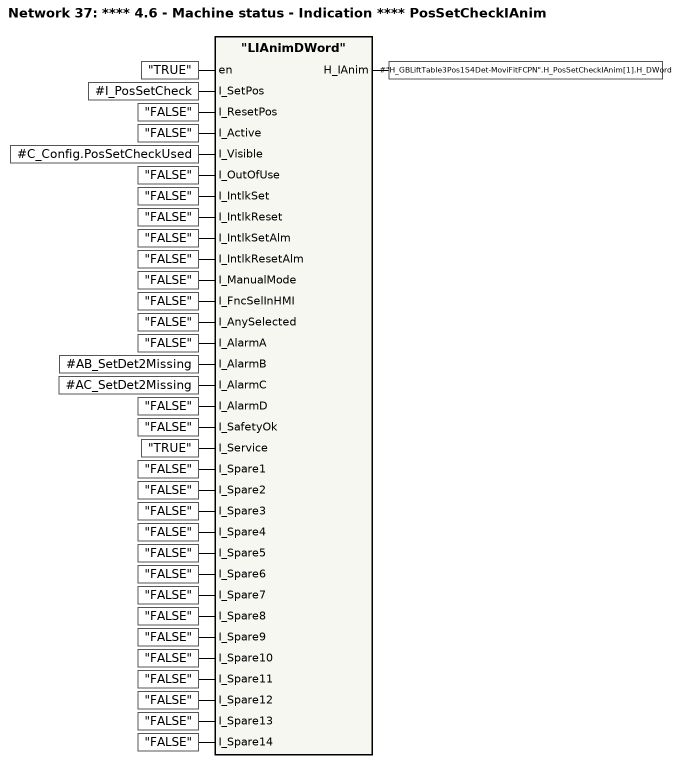
   IF "TRUE" THEN
       "LIAnimDWord"(I_SetPos := #I_PosSetCheck,
                     I_ResetPos := "FALSE",
                     I_Active := "FALSE",
                     I_Visible := #C_Config.PosSetCheckUsed,
                     I_OutOfUse := "FALSE",
                     I_IntlkSet := "FALSE",
                     I_IntlkReset := "FALSE",
                     I_IntlkSetAlm := "FALSE",
                     I_IntlkResetAlm := "FALSE",
                     I_ManualMode := "FALSE",
                     I_FncSelInHMI := "FALSE",
                     I_AnySelected := "FALSE",
                     I_AlarmA := "FALSE",
                     I_AlarmB := #AB_SetDet2Missing,
                     I_AlarmC := #AC_SetDet2Missing,
                     I_AlarmD := "FALSE",
                     I_SafetyOk := "FALSE",
                     I_Service := "TRUE",
                     I_Spare1 := "FALSE",
                     I_Spare2 := "FALSE",
                     I_Spare3 := "FALSE",
                     I_Spare4 := "FALSE",
                     I_Spare5 := "FALSE",
                     I_Spare6 := "FALSE",
                     I_Spare7 := "FALSE",
                     I_Spare8 := "FALSE",
                     I_Spare9 := "FALSE",
                     I_Spare10 := "FALSE",
                     I_Spare11 := "FALSE",
                     I_Spare12 := "FALSE",
                     I_Spare13 := "FALSE",
                     I_Spare14 := "FALSE",
                     H_IAnim => #"H_GBLiftTable3Pos1S4Det-MoviFitFCPN".H_PosSetCheckIAnim[1].H_DWord);
   END_IF;
END_REGION

REGION Network 38: **** 4.6 - Machine status - Indication **** PosMiddleIAnim
   // Icon animation
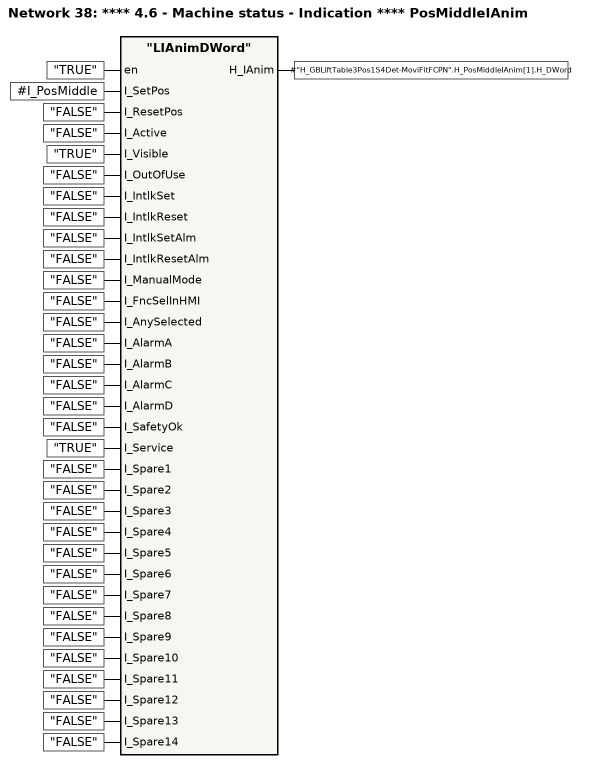
   IF "TRUE" THEN
       "LIAnimDWord"(I_SetPos := #I_PosMiddle,
                     I_ResetPos := "FALSE",
                     I_Active := "FALSE",
                     I_Visible := "TRUE",
                     I_OutOfUse := "FALSE",
                     I_IntlkSet := "FALSE",
                     I_IntlkReset := "FALSE",
                     I_IntlkSetAlm := "FALSE",
                     I_IntlkResetAlm := "FALSE",
                     I_ManualMode := "FALSE",
                     I_FncSelInHMI := "FALSE",
                     I_AnySelected := "FALSE",
                     I_AlarmA := "FALSE",
                     I_AlarmB := "FALSE",
                     I_AlarmC := "FALSE",
                     I_AlarmD := "FALSE",
                     I_SafetyOk := "FALSE",
                     I_Service := "TRUE",
                     I_Spare1 := "FALSE",
                     I_Spare2 := "FALSE",
                     I_Spare3 := "FALSE",
                     I_Spare4 := "FALSE",
                     I_Spare5 := "FALSE",
                     I_Spare6 := "FALSE",
                     I_Spare7 := "FALSE",
                     I_Spare8 := "FALSE",
                     I_Spare9 := "FALSE",
                     I_Spare10 := "FALSE",
                     I_Spare11 := "FALSE",
                     I_Spare12 := "FALSE",
                     I_Spare13 := "FALSE",
                     I_Spare14 := "FALSE",
                     H_IAnim => #"H_GBLiftTable3Pos1S4Det-MoviFitFCPN".H_PosMiddleIAnim[1].H_DWord);
   END_IF;
END_REGION

REGION Network 39: **** 4.6 - Machine status - Indication **** PosResIAnim
   // Icon animation
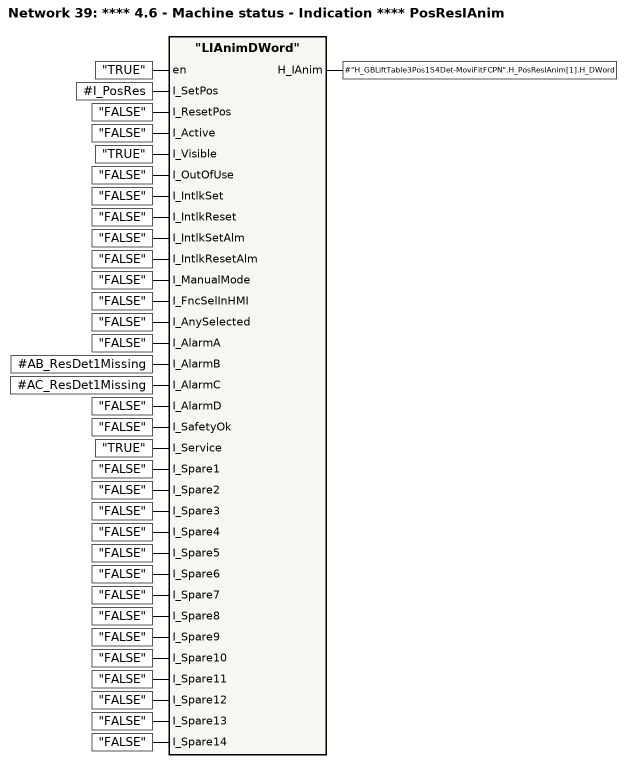
   IF "TRUE" THEN
       "LIAnimDWord"(I_SetPos := #I_PosRes,
                     I_ResetPos := "FALSE",
                     I_Active := "FALSE",
                     I_Visible := "TRUE",
                     I_OutOfUse := "FALSE",
                     I_IntlkSet := "FALSE",
                     I_IntlkReset := "FALSE",
                     I_IntlkSetAlm := "FALSE",
                     I_IntlkResetAlm := "FALSE",
                     I_ManualMode := "FALSE",
                     I_FncSelInHMI := "FALSE",
                     I_AnySelected := "FALSE",
                     I_AlarmA := "FALSE",
                     I_AlarmB := #AB_ResDet1Missing,
                     I_AlarmC := #AC_ResDet1Missing,
                     I_AlarmD := "FALSE",
                     I_SafetyOk := "FALSE",
                     I_Service := "TRUE",
                     I_Spare1 := "FALSE",
                     I_Spare2 := "FALSE",
                     I_Spare3 := "FALSE",
                     I_Spare4 := "FALSE",
                     I_Spare5 := "FALSE",
                     I_Spare6 := "FALSE",
                     I_Spare7 := "FALSE",
                     I_Spare8 := "FALSE",
                     I_Spare9 := "FALSE",
                     I_Spare10 := "FALSE",
                     I_Spare11 := "FALSE",
                     I_Spare12 := "FALSE",
                     I_Spare13 := "FALSE",
                     I_Spare14 := "FALSE",
                     H_IAnim => #"H_GBLiftTable3Pos1S4Det-MoviFitFCPN".H_PosResIAnim[1].H_DWord);
   END_IF;
END_REGION

REGION Network 40: **** 4.6 - Machine status - Indication **** PosResCheckIAnim
   // Icon animation
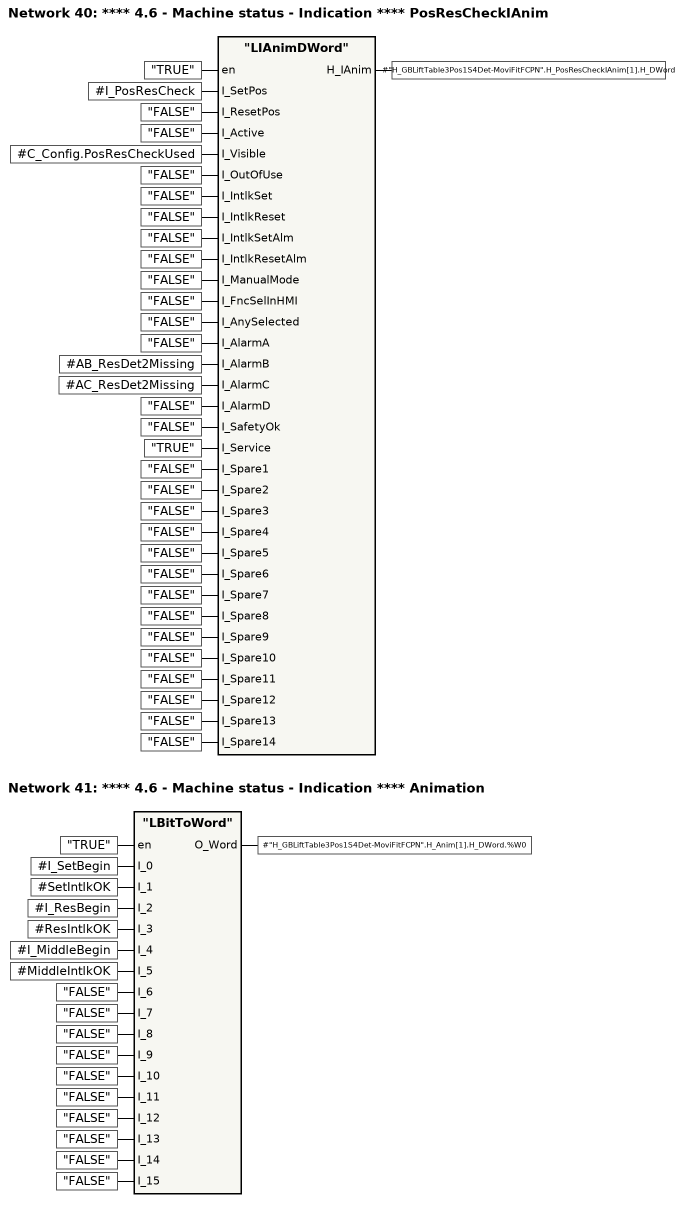
   IF "TRUE" THEN
       "LIAnimDWord"(I_SetPos := #I_PosResCheck,
                     I_ResetPos := "FALSE",
                     I_Active := "FALSE",
                     I_Visible := #C_Config.PosResCheckUsed,
                     I_OutOfUse := "FALSE",
                     I_IntlkSet := "FALSE",
                     I_IntlkReset := "FALSE",
                     I_IntlkSetAlm := "FALSE",
                     I_IntlkResetAlm := "FALSE",
                     I_ManualMode := "FALSE",
                     I_FncSelInHMI := "FALSE",
                     I_AnySelected := "FALSE",
                     I_AlarmA := "FALSE",
                     I_AlarmB := #AB_ResDet2Missing,
                     I_AlarmC := #AC_ResDet2Missing,
                     I_AlarmD := "FALSE",
                     I_SafetyOk := "FALSE",
                     I_Service := "TRUE",
                     I_Spare1 := "FALSE",
                     I_Spare2 := "FALSE",
                     I_Spare3 := "FALSE",
                     I_Spare4 := "FALSE",
                     I_Spare5 := "FALSE",
                     I_Spare6 := "FALSE",
                     I_Spare7 := "FALSE",
                     I_Spare8 := "FALSE",
                     I_Spare9 := "FALSE",
                     I_Spare10 := "FALSE",
                     I_Spare11 := "FALSE",
                     I_Spare12 := "FALSE",
                     I_Spare13 := "FALSE",
                     I_Spare14 := "FALSE",
                     H_IAnim => #"H_GBLiftTable3Pos1S4Det-MoviFitFCPN".H_PosResCheckIAnim[1].H_DWord);
   END_IF;
END_REGION

REGION Network 41: **** 4.6 - Machine status - Indication **** Animation
   // Animation
   IF "TRUE" THEN
       "LBitToWord"(I_0 := #I_SetBegin,
                    I_1 := #SetIntlkOK,
                    I_2 := #I_ResBegin,
                    I_3 := #ResIntlkOK,
                    I_4 := #I_MiddleBegin,
                    I_5 := #MiddleIntlkOK,
                    I_6 := "FALSE",
                    I_7 := "FALSE",
                    I_8 := "FALSE",
                    I_9 := "FALSE",
                    I_10 := "FALSE",
                    I_11 := "FALSE",
                    I_12 := "FALSE",
                    I_13 := "FALSE",
                    I_14 := "FALSE",
                    I_15 := "FALSE",
                    O_Word => #"H_GBLiftTable3Pos1S4Det-MoviFitFCPN".H_Anim[1].H_DWord.%W0);
   END_IF;
END_REGION

REGION Network 42: **** 4.6 - Machine status - Indication **** Animation
   // Animation
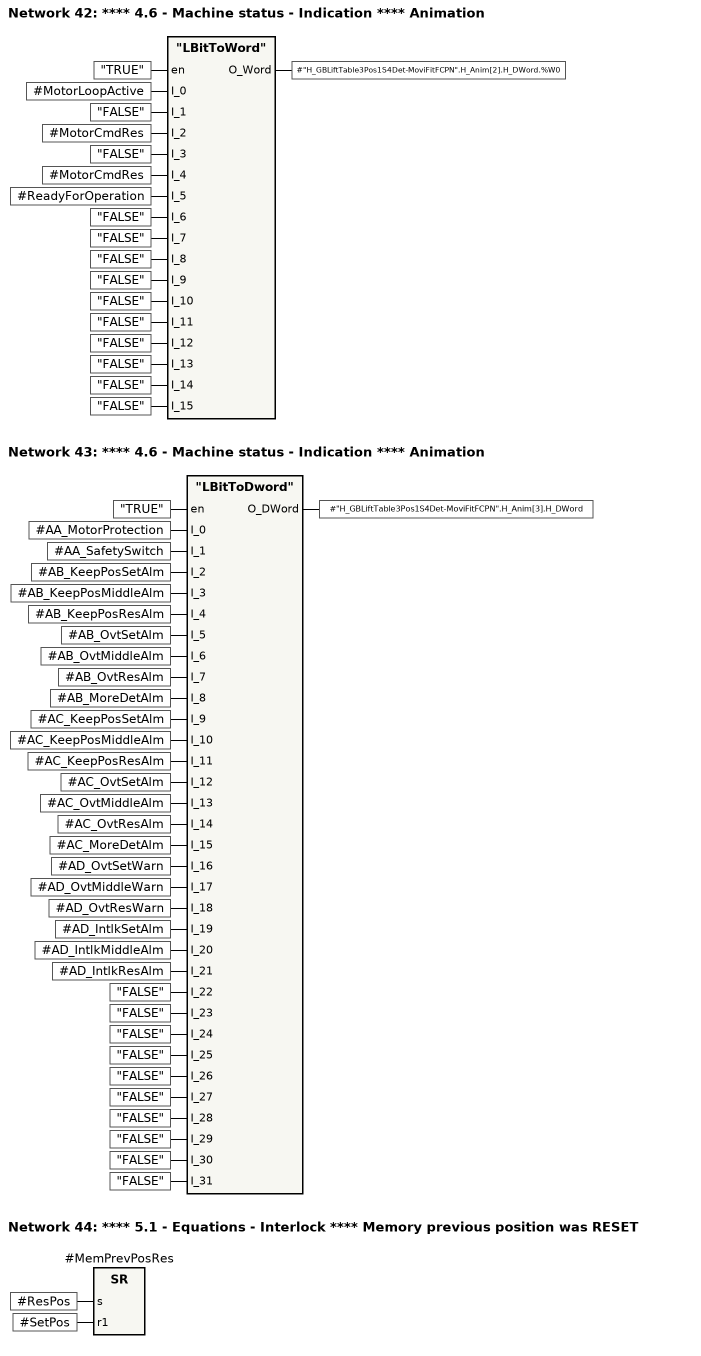
   IF "TRUE" THEN
       "LBitToWord"(I_0 := #MotorLoopActive,
                    I_1 := "FALSE",
                    I_2 := #MotorCmdRes,
                    I_3 := "FALSE",
                    I_4 := #MotorCmdRes,
                    I_5 := #ReadyForOperation,
                    I_6 := "FALSE",
                    I_7 := "FALSE",
                    I_8 := "FALSE",
                    I_9 := "FALSE",
                    I_10 := "FALSE",
                    I_11 := "FALSE",
                    I_12 := "FALSE",
                    I_13 := "FALSE",
                    I_14 := "FALSE",
                    I_15 := "FALSE",
                    O_Word => #"H_GBLiftTable3Pos1S4Det-MoviFitFCPN".H_Anim[2].H_DWord.%W0);
   END_IF;
END_REGION

REGION Network 43: **** 4.6 - Machine status - Indication **** Animation
   // Animation
   IF "TRUE" THEN
       "LBitToDword"(I_0 := #AA_MotorProtection,
                     I_1 := #AA_SafetySwitch,
                     I_2 := #AB_KeepPosSetAlm,
                     I_3 := #AB_KeepPosMiddleAlm,
                     I_4 := #AB_KeepPosResAlm,
                     I_5 := #AB_OvtSetAlm,
                     I_6 := #AB_OvtMiddleAlm,
                     I_7 := #AB_OvtResAlm,
                     I_8 := #AB_MoreDetAlm,
                     I_9 := #AC_KeepPosSetAlm,
                     I_10 := #AC_KeepPosMiddleAlm,
                     I_11 := #AC_KeepPosResAlm,
                     I_12 := #AC_OvtSetAlm,
                     I_13 := #AC_OvtMiddleAlm,
                     I_14 := #AC_OvtResAlm,
                     I_15 := #AC_MoreDetAlm,
                     I_16 := #AD_OvtSetWarn,
                     I_17 := #AD_OvtMiddleWarn,
                     I_18 := #AD_OvtResWarn,
                     I_19 := #AD_IntlkSetAlm,
                     I_20 := #AD_IntlkMiddleAlm,
                     I_21 := #AD_IntlkResAlm,
                     I_22 := "FALSE",
                     I_23 := "FALSE",
                     I_24 := "FALSE",
                     I_25 := "FALSE",
                     I_26 := "FALSE",
                     I_27 := "FALSE",
                     I_28 := "FALSE",
                     I_29 := "FALSE",
                     I_30 := "FALSE",
                     I_31 := "FALSE",
                     O_DWord => #"H_GBLiftTable3Pos1S4Det-MoviFitFCPN".H_Anim[3].H_DWord);
   END_IF;
END_REGION

REGION Network 44: **** 5.1 - Equations - Interlock **** Memory previous position was RESET
   // Memory previous position was RESET
   IF #ResPos THEN
       #MemPrevPosRes := TRUE;   // SR flip-flop
   END_IF;
   IF #SetPos THEN #MemPrevPosRes := FALSE; END_IF;
END_REGION

REGION Network 45: **** 5.1 - Equations **** Motor Command Set
   // Command Set
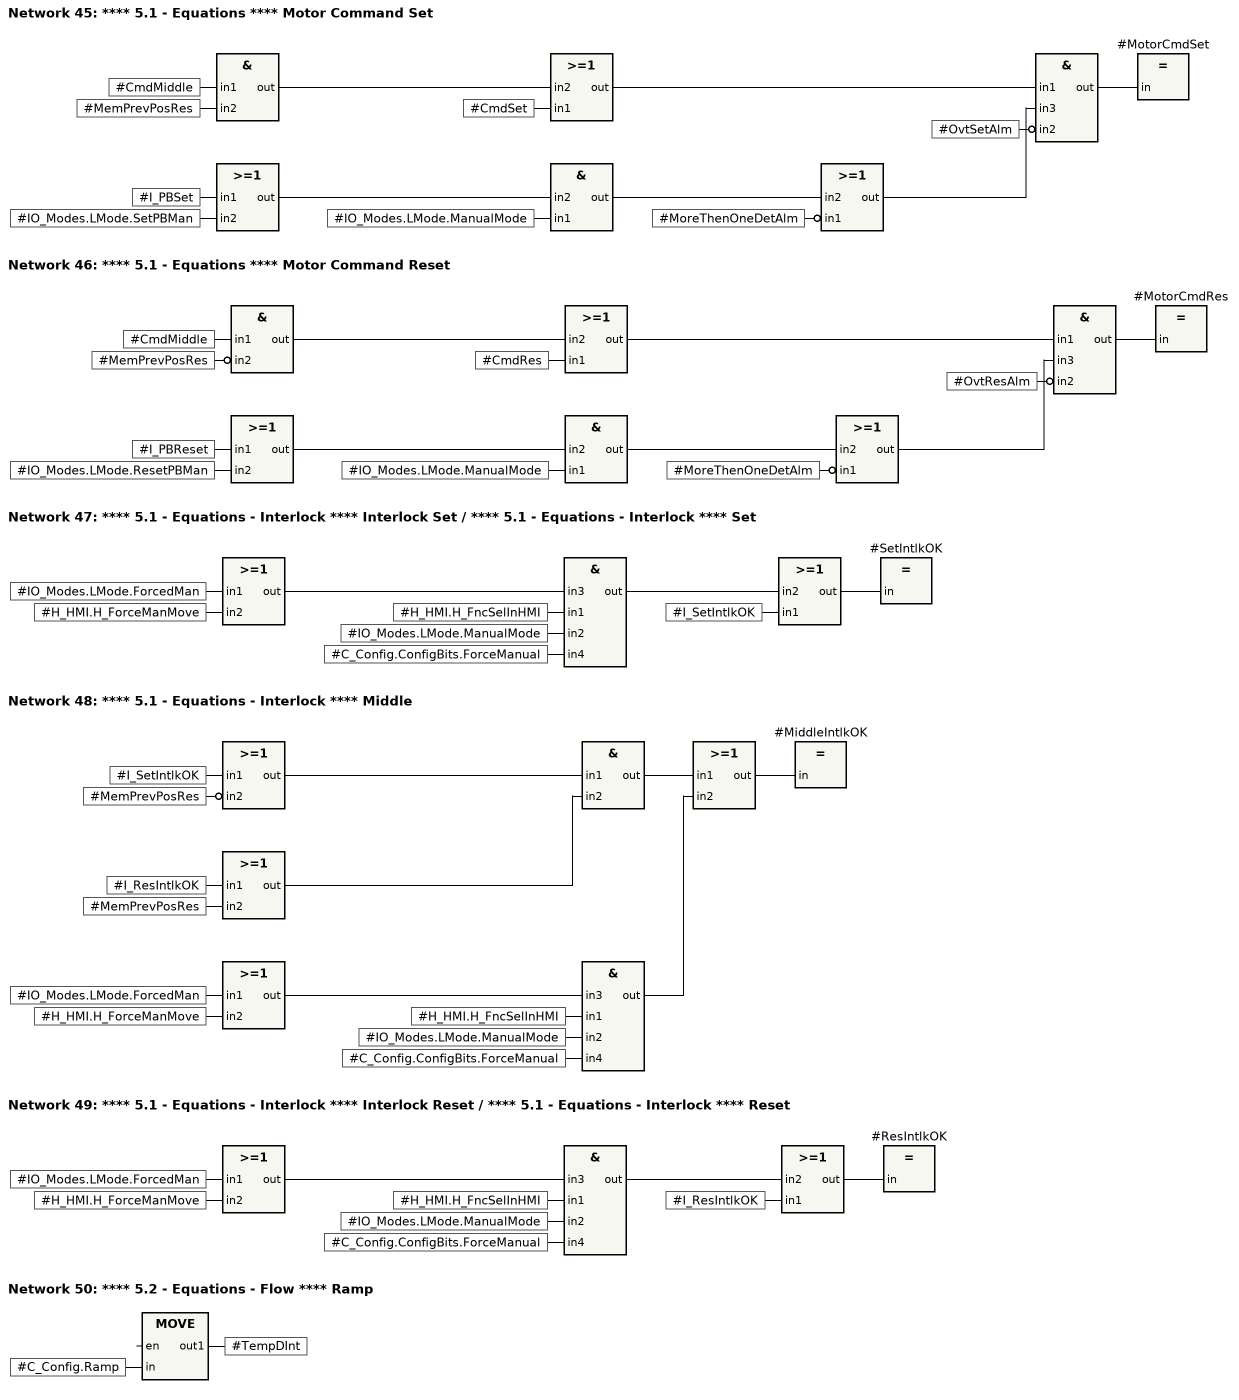
   #MotorCmdSet := ((#CmdMiddle AND #MemPrevPosRes) OR #CmdSet) AND (((#I_PBSet OR #IO_Modes.LMode.SetPBMan) AND #IO_Modes.LMode.ManualMode) OR NOT #MoreThenOneDetAlm) AND NOT #OvtSetAlm;
END_REGION

REGION Network 46: **** 5.1 - Equations **** Motor Command Reset
   // Command Reset
   #MotorCmdRes := ((#CmdMiddle AND NOT #MemPrevPosRes) OR #CmdRes) AND (((#I_PBReset OR #IO_Modes.LMode.ResetPBMan) AND #IO_Modes.LMode.ManualMode) OR NOT #MoreThenOneDetAlm) AND NOT #OvtResAlm;
END_REGION

REGION Network 47: **** 5.1 - Equations - Interlock **** Interlock Set / **** 5.1 - Equations - Interlock **** Set
   // Interlock
   #SetIntlkOK := ((#IO_Modes.LMode.ForcedMan OR #H_HMI.H_ForceManMove) AND #H_HMI.H_FncSelInHMI AND #IO_Modes.LMode.ManualMode AND #C_Config.ConfigBits.ForceManual) OR #I_SetIntlkOK;
END_REGION

REGION Network 48: **** 5.1 - Equations - Interlock **** Middle
   // Interlock
   #MiddleIntlkOK := ((#I_SetIntlkOK OR NOT #MemPrevPosRes) AND (#I_ResIntlkOK OR #MemPrevPosRes)) OR ((#IO_Modes.LMode.ForcedMan OR #H_HMI.H_ForceManMove) AND #H_HMI.H_FncSelInHMI AND #IO_Modes.LMode.ManualMode AND #C_Config.ConfigBits.ForceManual);
END_REGION

REGION Network 49: **** 5.1 - Equations - Interlock **** Interlock Reset / **** 5.1 - Equations - Interlock **** Reset
   // Interlock
   #ResIntlkOK := ((#IO_Modes.LMode.ForcedMan OR #H_HMI.H_ForceManMove) AND #H_HMI.H_FncSelInHMI AND #IO_Modes.LMode.ManualMode AND #C_Config.ConfigBits.ForceManual) OR #I_ResIntlkOK;
END_REGION

REGION Network 50: **** 5.2 - Equations - Flow **** Ramp
   #TempDInt := #C_Config.Ramp;
END_REGION

REGION Network 51: **** 5.1 - Equations **** Start Movement to middle
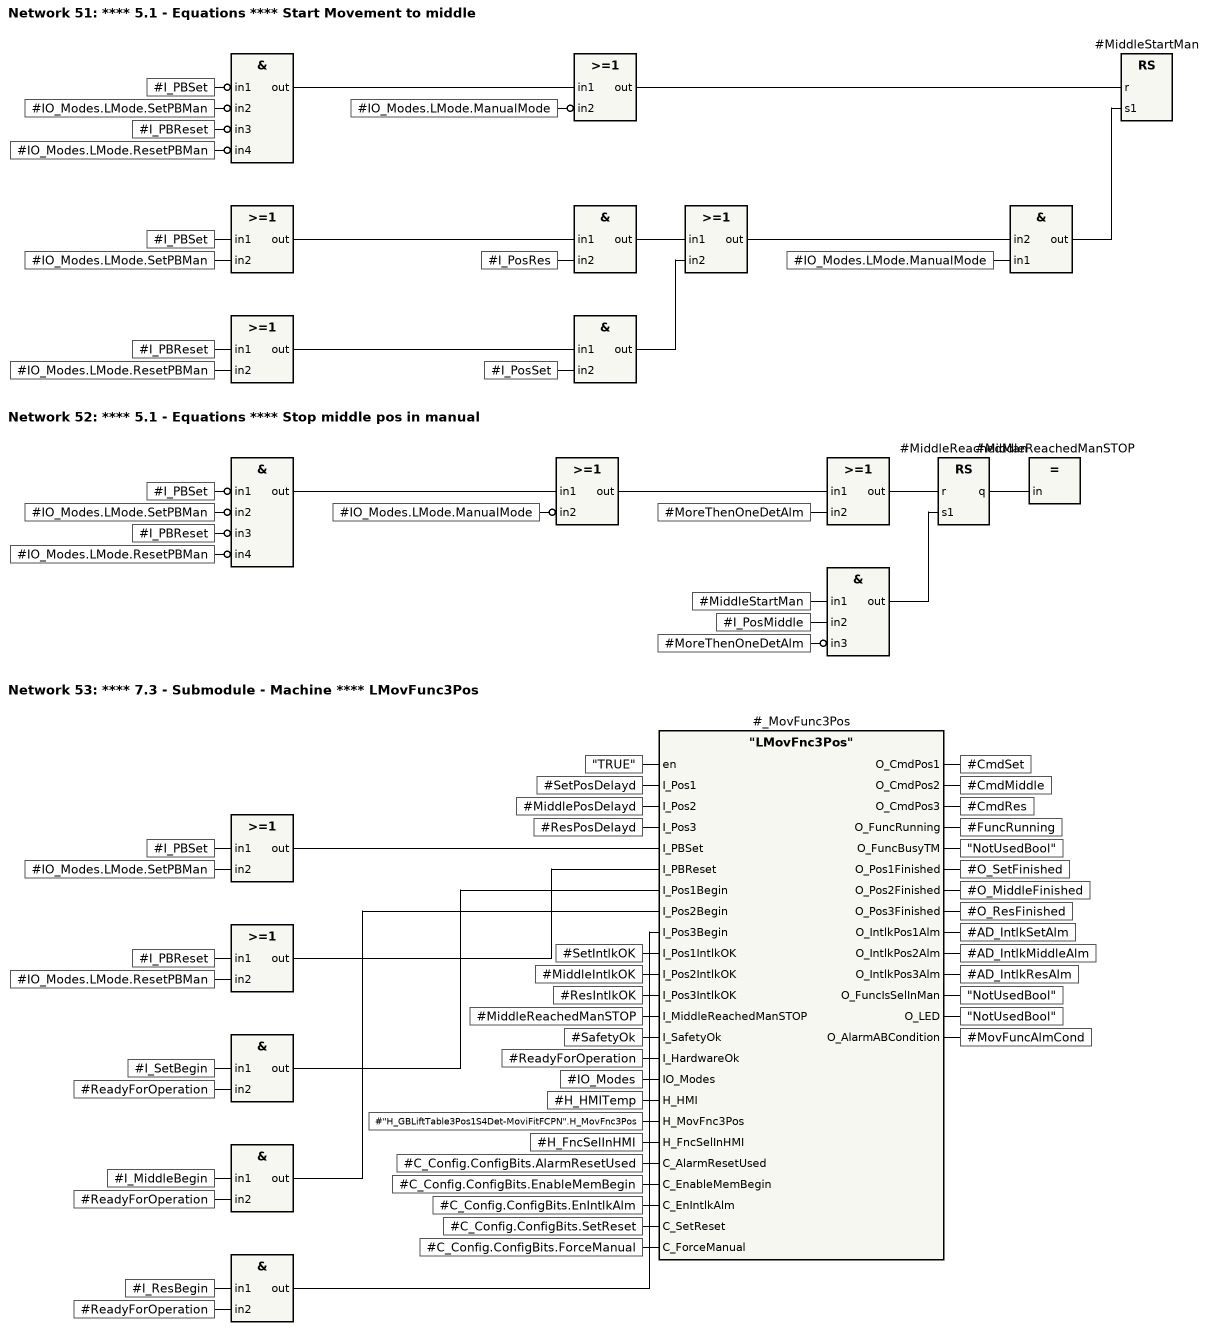
   IF (NOT #I_PBSet AND NOT #IO_Modes.LMode.SetPBMan AND NOT #I_PBReset AND NOT #IO_Modes.LMode.ResetPBMan) OR NOT #IO_Modes.LMode.ManualMode THEN
       #MiddleStartMan := FALSE;   // RS flip-flop
   END_IF;
   IF (((#I_PBSet OR #IO_Modes.LMode.SetPBMan) AND #I_PosRes) OR ((#I_PBReset OR #IO_Modes.LMode.ResetPBMan) AND #I_PosSet)) AND #IO_Modes.LMode.ManualMode THEN
       #MiddleStartMan := TRUE;
   END_IF;
END_REGION

REGION Network 52: **** 5.1 - Equations **** Stop middle pos in manual
   IF (NOT #I_PBSet AND NOT #IO_Modes.LMode.SetPBMan AND NOT #I_PBReset AND NOT #IO_Modes.LMode.ResetPBMan) OR NOT #IO_Modes.LMode.ManualMode OR #MoreThenOneDetAlm THEN
       #MiddleReachedMan := FALSE;   // RS flip-flop
   END_IF;
   IF #MiddleStartMan AND #I_PosMiddle AND NOT #MoreThenOneDetAlm THEN #MiddleReachedMan := TRUE; END_IF;
   #MiddleReachedManSTOP := #MiddleReachedMan;
END_REGION

REGION Network 53: **** 7.3 - Submodule - Machine **** LMovFunc3Pos
   // LMovFunc2Pos / LMovFunc3Pos
   IF "TRUE" THEN
       #_MovFunc3Pos(I_Pos1 := #SetPosDelayd,   // "LMovFnc3Pos"
                     I_Pos2 := #MiddlePosDelayd,
                     I_Pos3 := #ResPosDelayd,
                     I_PBSet := #I_PBSet OR #IO_Modes.LMode.SetPBMan,
                     I_PBReset := #I_PBReset OR #IO_Modes.LMode.ResetPBMan,
                     I_Pos1Begin := #I_SetBegin AND #ReadyForOperation,
                     I_Pos2Begin := #I_MiddleBegin AND #ReadyForOperation,
                     I_Pos3Begin := #I_ResBegin AND #ReadyForOperation,
                     I_Pos1IntlkOK := #SetIntlkOK,
                     I_Pos2IntlkOK := #MiddleIntlkOK,
                     I_Pos3IntlkOK := #ResIntlkOK,
                     I_MiddleReachedManSTOP := #MiddleReachedManSTOP,
                     I_SafetyOk := #SafetyOk,
                     I_HardwareOk := #ReadyForOperation,
                     IO_Modes := #IO_Modes,
                     H_HMI := #H_HMITemp,
                     H_MovFnc3Pos := #"H_GBLiftTable3Pos1S4Det-MoviFitFCPN".H_MovFnc3Pos,
                     H_FncSelInHMI := #H_FncSelInHMI,
                     C_AlarmResetUsed := #C_Config.ConfigBits.AlarmResetUsed,
                     C_EnableMemBegin := #C_Config.ConfigBits.EnableMemBegin,
                     C_EnIntlkAlm := #C_Config.ConfigBits.EnIntlkAlm,
                     C_SetReset := #C_Config.ConfigBits.SetReset,
                     C_ForceManual := #C_Config.ConfigBits.ForceManual,
                     O_CmdPos1 => #CmdSet,
                     O_CmdPos2 => #CmdMiddle,
                     O_CmdPos3 => #CmdRes,
                     O_FuncRunning => #FuncRunning,
                     O_FuncBusyTM => "NotUsedBool",
                     O_Pos1Finished => #O_SetFinished,
                     O_Pos2Finished => #O_MiddleFinished,
                     O_Pos3Finished => #O_ResFinished,
                     O_IntlkPos1Alm => #AD_IntlkSetAlm,
                     O_IntlkPos2Alm => #AD_IntlkMiddleAlm,
                     O_IntlkPos3Alm => #AD_IntlkResAlm,
                     O_FuncIsSelInMan => "NotUsedBool",
                     O_LED => "NotUsedBool",
                     O_AlarmABCondition => #MovFuncAlmCond);
   END_IF;
END_REGION

REGION Network 54: **** 7.3 - Submodule - Machine **** LMovFunc3Pos Move UDT
   // LMovFunc3Pos Move UDT
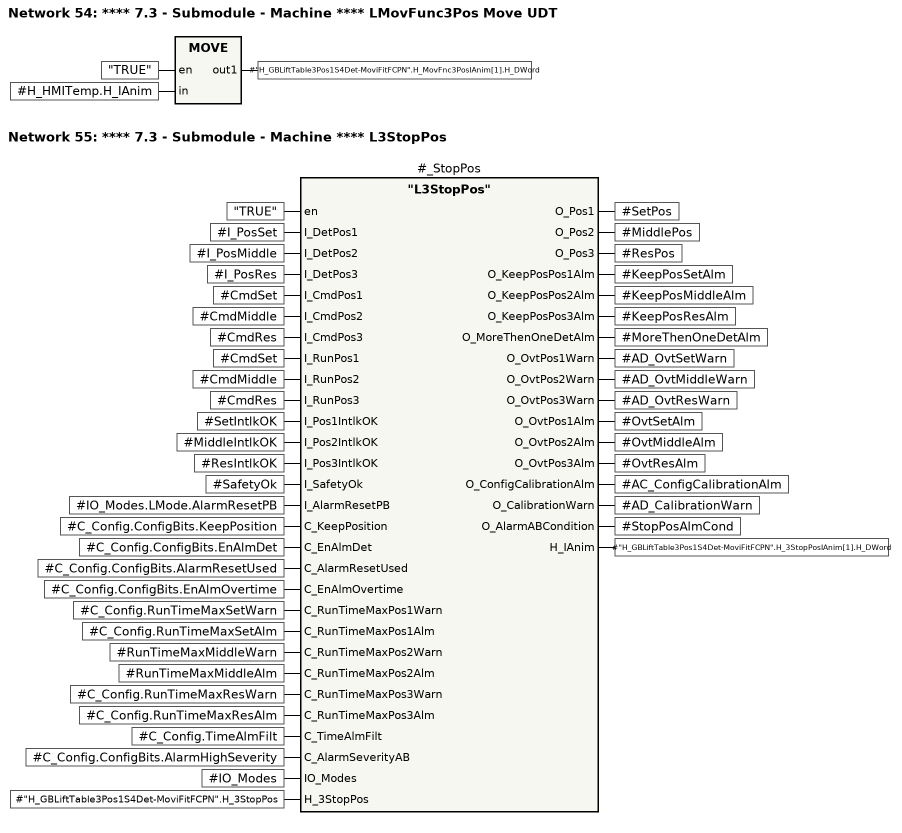
   IF "TRUE" THEN
       #"H_GBLiftTable3Pos1S4Det-MoviFitFCPN".H_MovFnc3PosIAnim[1].H_DWord := #H_HMITemp.H_IAnim;
   END_IF;
END_REGION

REGION Network 55: **** 7.3 - Submodule - Machine **** L3StopPos
   // L3StopPos
   IF "TRUE" THEN
       #_StopPos(I_DetPos1 := #I_PosSet,   // "L3StopPos"
                 I_DetPos2 := #I_PosMiddle,
                 I_DetPos3 := #I_PosRes,
                 I_CmdPos1 := #CmdSet,
                 I_CmdPos2 := #CmdMiddle,
                 I_CmdPos3 := #CmdRes,
                 I_RunPos1 := #CmdSet,
                 I_RunPos2 := #CmdMiddle,
                 I_RunPos3 := #CmdRes,
                 I_Pos1IntlkOK := #SetIntlkOK,
                 I_Pos2IntlkOK := #MiddleIntlkOK,
                 I_Pos3IntlkOK := #ResIntlkOK,
                 I_SafetyOk := #SafetyOk,
                 I_AlarmResetPB := #IO_Modes.LMode.AlarmResetPB,
                 C_KeepPosition := #C_Config.ConfigBits.KeepPosition,
                 C_EnAlmDet := #C_Config.ConfigBits.EnAlmDet,
                 C_AlarmResetUsed := #C_Config.ConfigBits.AlarmResetUsed,
                 C_EnAlmOvertime := #C_Config.ConfigBits.EnAlmOvertime,
                 C_RunTimeMaxPos1Warn := #C_Config.RunTimeMaxSetWarn,
                 C_RunTimeMaxPos1Alm := #C_Config.RunTimeMaxSetAlm,
                 C_RunTimeMaxPos2Warn := #RunTimeMaxMiddleWarn,
                 C_RunTimeMaxPos2Alm := #RunTimeMaxMiddleAlm,
                 C_RunTimeMaxPos3Warn := #C_Config.RunTimeMaxResWarn,
                 C_RunTimeMaxPos3Alm := #C_Config.RunTimeMaxResAlm,
                 C_TimeAlmFilt := #C_Config.TimeAlmFilt,
                 C_AlarmSeverityAB := #C_Config.ConfigBits.AlarmHighSeverity,
                 IO_Modes := #IO_Modes,
                 H_3StopPos := #"H_GBLiftTable3Pos1S4Det-MoviFitFCPN".H_3StopPos,
                 O_Pos1 => #SetPos,
                 O_Pos2 => #MiddlePos,
                 O_Pos3 => #ResPos,
                 O_KeepPosPos1Alm => #KeepPosSetAlm,
                 O_KeepPosPos2Alm => #KeepPosMiddleAlm,
                 O_KeepPosPos3Alm => #KeepPosResAlm,
                 O_MoreThenOneDetAlm => #MoreThenOneDetAlm,
                 O_OvtPos1Warn => #AD_OvtSetWarn,
                 O_OvtPos2Warn => #AD_OvtMiddleWarn,
                 O_OvtPos3Warn => #AD_OvtResWarn,
                 O_OvtPos1Alm => #OvtSetAlm,
                 O_OvtPos2Alm => #OvtMiddleAlm,
                 O_OvtPos3Alm => #OvtResAlm,
                 O_ConfigCalibrationAlm => #AC_ConfigCalibrationAlm,
                 O_CalibrationWarn => #AD_CalibrationWarn,
                 O_AlarmABCondition => #StopPosAlmCond,
                 H_IAnim => #"H_GBLiftTable3Pos1S4Det-MoviFitFCPN".H_3StopPosIAnim[1].H_DWord);
   END_IF;
END_REGION

REGION Network 56: **** 7.3 - Submodule - Machine **** Motor Loop MOVIFIT-FC
   // Motor loop G120
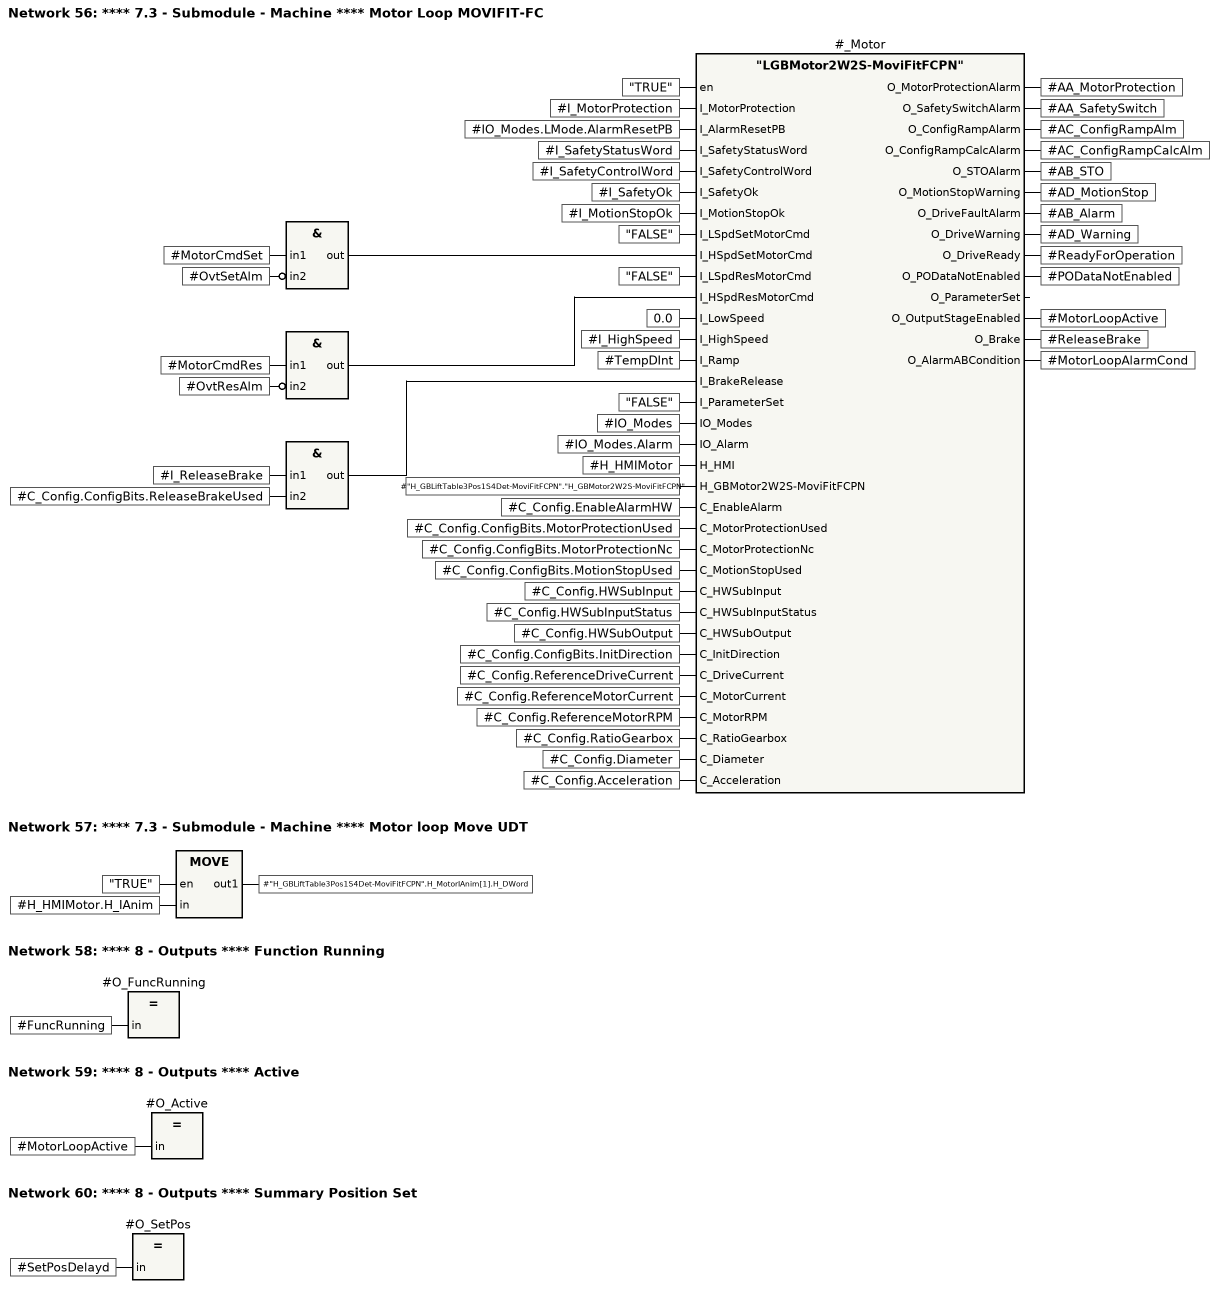
   IF "TRUE" THEN
       #_Motor(I_MotorProtection := #I_MotorProtection,   // "LGBMotor2W2S-MoviFitFCPN"
               I_AlarmResetPB := #IO_Modes.LMode.AlarmResetPB,
               I_SafetyStatusWord := #I_SafetyStatusWord,
               I_SafetyControlWord := #I_SafetyControlWord,
               I_SafetyOk := #I_SafetyOk,
               I_MotionStopOk := #I_MotionStopOk,
               I_LSpdSetMotorCmd := "FALSE",
               I_HSpdSetMotorCmd := #MotorCmdSet AND NOT #OvtSetAlm,
               I_LSpdResMotorCmd := "FALSE",
               I_HSpdResMotorCmd := #MotorCmdRes AND NOT #OvtResAlm,
               I_LowSpeed := 0.0,
               I_HighSpeed := #I_HighSpeed,
               I_Ramp := #TempDInt,
               I_BrakeRelease := #I_ReleaseBrake AND #C_Config.ConfigBits.ReleaseBrakeUsed,
               I_ParameterSet := "FALSE",
               IO_Modes := #IO_Modes,
               IO_Alarm := #IO_Modes.Alarm,
               H_HMI := #H_HMIMotor,
               "H_GBMotor2W2S-MoviFitFCPN" := #"H_GBLiftTable3Pos1S4Det-MoviFitFCPN"."H_GBMotor2W2S-MoviFitFCPN",
               C_EnableAlarm := #C_Config.EnableAlarmHW,
               C_MotorProtectionUsed := #C_Config.ConfigBits.MotorProtectionUsed,
               C_MotorProtectionNc := #C_Config.ConfigBits.MotorProtectionNc,
               C_MotionStopUsed := #C_Config.ConfigBits.MotionStopUsed,
               C_HWSubInput := #C_Config.HWSubInput,
               C_HWSubInputStatus := #C_Config.HWSubInputStatus,
               C_HWSubOutput := #C_Config.HWSubOutput,
               C_InitDirection := #C_Config.ConfigBits.InitDirection,
               C_DriveCurrent := #C_Config.ReferenceDriveCurrent,
               C_MotorCurrent := #C_Config.ReferenceMotorCurrent,
               C_MotorRPM := #C_Config.ReferenceMotorRPM,
               C_RatioGearbox := #C_Config.RatioGearbox,
               C_Diameter := #C_Config.Diameter,
               C_Acceleration := #C_Config.Acceleration,
               O_MotorProtectionAlarm => #AA_MotorProtection,
               O_SafetySwitchAlarm => #AA_SafetySwitch,
               O_ConfigRampAlarm => #AC_ConfigRampAlm,
               O_ConfigRampCalcAlarm => #AC_ConfigRampCalcAlm,
               O_STOAlarm => #AB_STO,
               O_MotionStopWarning => #AD_MotionStop,
               O_DriveFaultAlarm => #AB_Alarm,
               O_DriveWarning => #AD_Warning,
               O_DriveReady => #ReadyForOperation,
               O_PODataNotEnabled => #PODataNotEnabled,
               O_OutputStageEnabled => #MotorLoopActive,
               O_Brake => #ReleaseBrake,
               O_AlarmABCondition => #MotorLoopAlarmCond);
   END_IF;
END_REGION

REGION Network 57: **** 7.3 - Submodule - Machine **** Motor loop Move UDT
   IF "TRUE" THEN
       #"H_GBLiftTable3Pos1S4Det-MoviFitFCPN".H_MotorIAnim[1].H_DWord := #H_HMIMotor.H_IAnim;
   END_IF;
END_REGION

REGION Network 58: **** 8 - Outputs **** Function Running
   // Function Running
   #O_FuncRunning := #FuncRunning;
END_REGION

REGION Network 59: **** 8 - Outputs **** Active
   // Motor Loop active
   #O_Active := #MotorLoopActive;
END_REGION

REGION Network 60: **** 8 - Outputs **** Summary Position Set
   // Summary Position Set
   #O_SetPos := #SetPosDelayd;
END_REGION

REGION Network 61: **** 8 - Outputs **** Summary Position Middle
   // Summary Position Middle
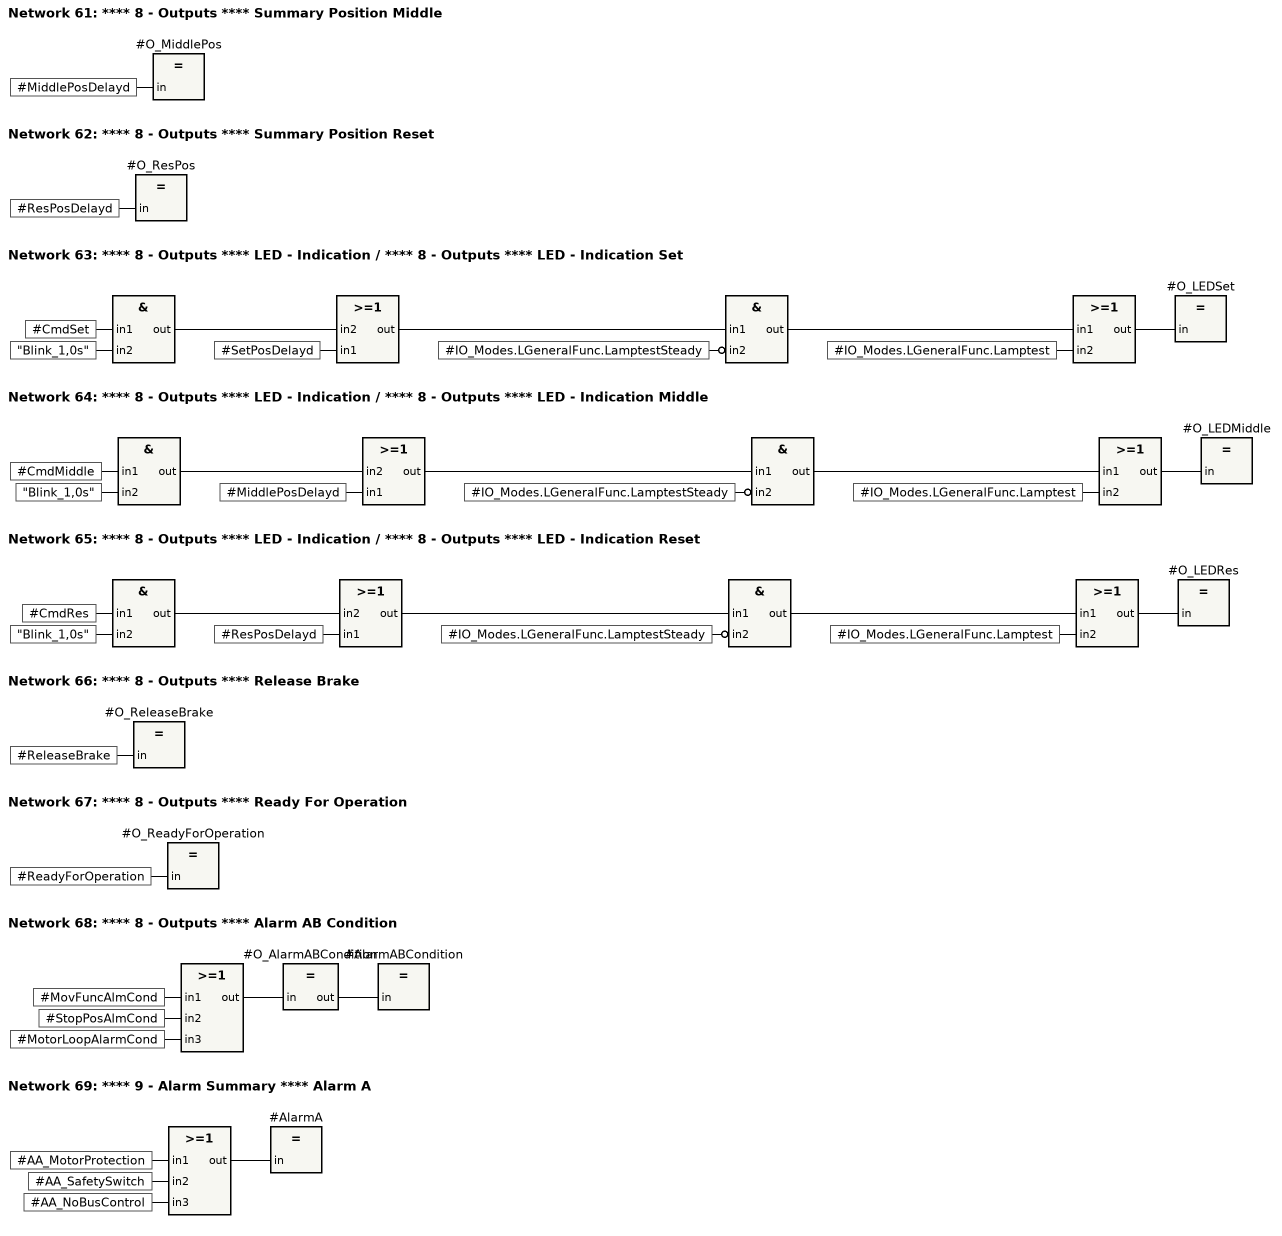
   #O_MiddlePos := #MiddlePosDelayd;
END_REGION

REGION Network 62: **** 8 - Outputs **** Summary Position Reset
   // Summary Position Reset
   #O_ResPos := #ResPosDelayd;
END_REGION

REGION Network 63: **** 8 - Outputs **** LED - Indication / **** 8 - Outputs **** LED - Indication Set
   // LED - Indication
   #O_LEDSet := (((#CmdSet AND "Blink_1,0s") OR #SetPosDelayd) AND NOT #IO_Modes.LGeneralFunc.LamptestSteady) OR #IO_Modes.LGeneralFunc.Lamptest;
END_REGION

REGION Network 64: **** 8 - Outputs **** LED - Indication / **** 8 - Outputs **** LED - Indication Middle
   // LED - Indication
   #O_LEDMiddle := (((#CmdMiddle AND "Blink_1,0s") OR #MiddlePosDelayd) AND NOT #IO_Modes.LGeneralFunc.LamptestSteady) OR #IO_Modes.LGeneralFunc.Lamptest;
END_REGION

REGION Network 65: **** 8 - Outputs **** LED - Indication / **** 8 - Outputs **** LED - Indication Reset
   // LED - Indication
   #O_LEDRes := (((#CmdRes AND "Blink_1,0s") OR #ResPosDelayd) AND NOT #IO_Modes.LGeneralFunc.LamptestSteady) OR #IO_Modes.LGeneralFunc.Lamptest;
END_REGION

REGION Network 66: **** 8 - Outputs **** Release Brake
   // Release Brake
   #O_ReleaseBrake := #ReleaseBrake;
END_REGION

REGION Network 67: **** 8 - Outputs **** Ready For Operation
   // Ready For Operation
   #O_ReadyForOperation := #ReadyForOperation;
END_REGION

REGION Network 68: **** 8 - Outputs **** Alarm AB Condition
   // Alarm AB condition
   #O_AlarmABCondition := #MovFuncAlmCond OR #StopPosAlmCond OR #MotorLoopAlarmCond;
   #AlarmABCondition := #O_AlarmABCondition;
END_REGION

REGION Network 69: **** 9 - Alarm Summary **** Alarm A
   // Alarms A
   #AlarmA := #AA_MotorProtection OR #AA_SafetySwitch OR #AA_NoBusControl;
END_REGION

REGION Network 70: **** 9 - Alarm Summary **** Alarm B
   // Alarms B
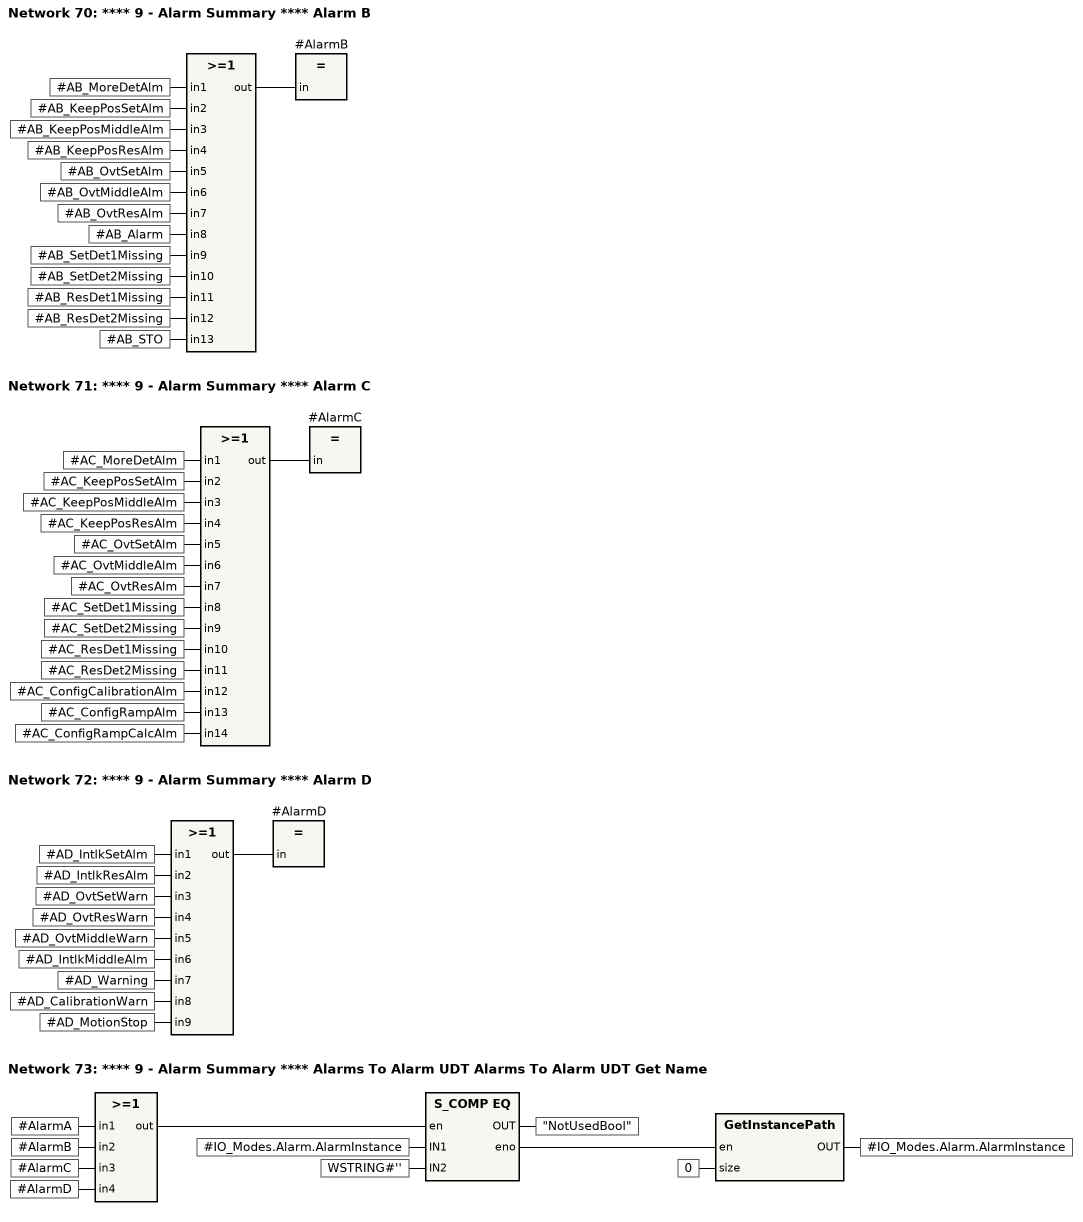
   #AlarmB := #AB_MoreDetAlm OR #AB_KeepPosSetAlm OR #AB_KeepPosMiddleAlm OR #AB_KeepPosResAlm OR #AB_OvtSetAlm OR #AB_OvtMiddleAlm OR #AB_OvtResAlm OR #AB_Alarm OR #AB_SetDet1Missing OR #AB_SetDet2Missing OR #AB_ResDet1Missing OR #AB_ResDet2Missing OR #AB_STO;
END_REGION

REGION Network 71: **** 9 - Alarm Summary **** Alarm C
   // Alarms C
   #AlarmC := #AC_MoreDetAlm OR #AC_KeepPosSetAlm OR #AC_KeepPosMiddleAlm OR #AC_KeepPosResAlm OR #AC_OvtSetAlm OR #AC_OvtMiddleAlm OR #AC_OvtResAlm OR #AC_SetDet1Missing OR #AC_SetDet2Missing OR #AC_ResDet1Missing OR #AC_ResDet2Missing OR #AC_ConfigCalibrationAlm OR #AC_ConfigRampAlm OR #AC_ConfigRampCalcAlm;
END_REGION

REGION Network 72: **** 9 - Alarm Summary **** Alarm D
   // Alarms D
   #AlarmD := #AD_IntlkSetAlm OR #AD_IntlkResAlm OR #AD_OvtSetWarn OR #AD_OvtResWarn OR #AD_OvtMiddleWarn OR #AD_IntlkMiddleAlm OR #AD_Warning OR #AD_CalibrationWarn OR #AD_MotionStop;
END_REGION

REGION Network 73: **** 9 - Alarm Summary **** Alarms To Alarm UDT Alarms To Alarm UDT Get Name
   // Alarm D
   S_COMP(EN := #AlarmA OR #AlarmB OR #AlarmC OR #AlarmD,
          IN1 := #IO_Modes.Alarm.AlarmInstance,
          IN2 := WSTRING#'',
          OUT => "NotUsedBool",
          ENO => #_w1);
   IF #_w1 THEN GetInstancePath(size := 0, OUT => #IO_Modes.Alarm.AlarmInstance); END_IF;
END_REGION

REGION Network 74: **** 9 - Alarm Summary **** Alarms To Alarm UDT
   // Alarm D
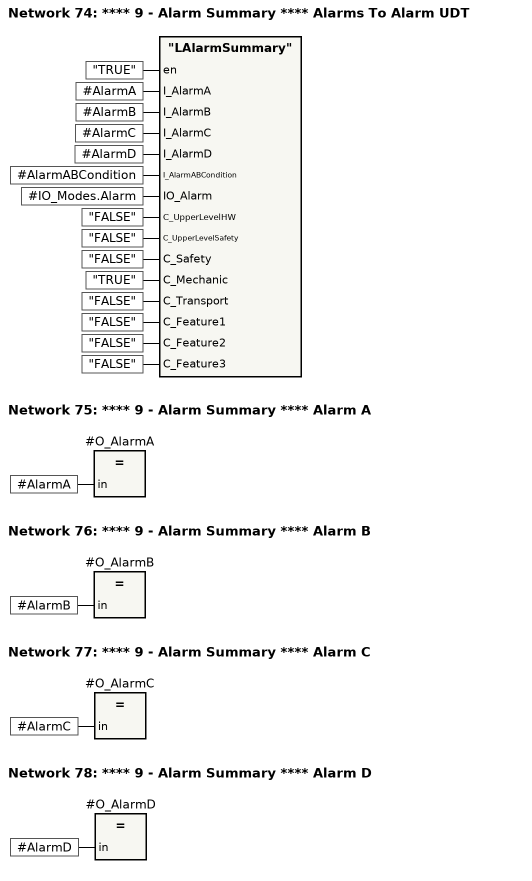
   IF "TRUE" THEN
       "LAlarmSummary"(I_AlarmA := #AlarmA,
                       I_AlarmB := #AlarmB,
                       I_AlarmC := #AlarmC,
                       I_AlarmD := #AlarmD,
                       I_AlarmABCondition := #AlarmABCondition,
                       IO_Alarm := #IO_Modes.Alarm,
                       C_UpperLevelHW := "FALSE",
                       C_UpperLevelSafety := "FALSE",
                       C_Safety := "FALSE",
                       C_Mechanic := "TRUE",
                       C_Transport := "FALSE",
                       C_Feature1 := "FALSE",
                       C_Feature2 := "FALSE",
                       C_Feature3 := "FALSE");
   END_IF;
END_REGION

REGION Network 75: **** 9 - Alarm Summary **** Alarm A
   // Alarm A
   #O_AlarmA := #AlarmA;
END_REGION

REGION Network 76: **** 9 - Alarm Summary **** Alarm B
   // Alarm B
   #O_AlarmB := #AlarmB;
END_REGION

REGION Network 77: **** 9 - Alarm Summary **** Alarm C
   // Alarm C
   #O_AlarmC := #AlarmC;
END_REGION

REGION Network 78: **** 9 - Alarm Summary **** Alarm D
   // Alarm D
   #O_AlarmD := #AlarmD;
END_REGION

REGION Network 79: **** 9 - Alarm Summary **** Alarm To Word
   // Alarm To Word
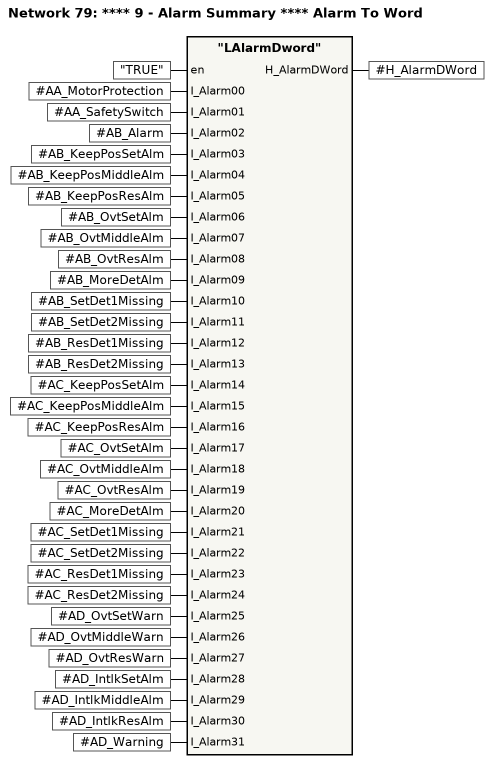
   IF "TRUE" THEN
       "LAlarmDword"(I_Alarm00 := #AA_MotorProtection,
                     I_Alarm01 := #AA_SafetySwitch,
                     I_Alarm02 := #AB_Alarm,
                     I_Alarm03 := #AB_KeepPosSetAlm,
                     I_Alarm04 := #AB_KeepPosMiddleAlm,
                     I_Alarm05 := #AB_KeepPosResAlm,
                     I_Alarm06 := #AB_OvtSetAlm,
                     I_Alarm07 := #AB_OvtMiddleAlm,
                     I_Alarm08 := #AB_OvtResAlm,
                     I_Alarm09 := #AB_MoreDetAlm,
                     I_Alarm10 := #AB_SetDet1Missing,
                     I_Alarm11 := #AB_SetDet2Missing,
                     I_Alarm12 := #AB_ResDet1Missing,
                     I_Alarm13 := #AB_ResDet2Missing,
                     I_Alarm14 := #AC_KeepPosSetAlm,
                     I_Alarm15 := #AC_KeepPosMiddleAlm,
                     I_Alarm16 := #AC_KeepPosResAlm,
                     I_Alarm17 := #AC_OvtSetAlm,
                     I_Alarm18 := #AC_OvtMiddleAlm,
                     I_Alarm19 := #AC_OvtResAlm,
                     I_Alarm20 := #AC_MoreDetAlm,
                     I_Alarm21 := #AC_SetDet1Missing,
                     I_Alarm22 := #AC_SetDet2Missing,
                     I_Alarm23 := #AC_ResDet1Missing,
                     I_Alarm24 := #AC_ResDet2Missing,
                     I_Alarm25 := #AD_OvtSetWarn,
                     I_Alarm26 := #AD_OvtMiddleWarn,
                     I_Alarm27 := #AD_OvtResWarn,
                     I_Alarm28 := #AD_IntlkSetAlm,
                     I_Alarm29 := #AD_IntlkMiddleAlm,
                     I_Alarm30 := #AD_IntlkResAlm,
                     I_Alarm31 := #AD_Warning,
                     H_AlarmDWord => #H_AlarmDWord);
   END_IF;
END_REGION

REGION Network 80: **** 9 - Alarm Summary **** Alarm To Word
   // Alarm To Word
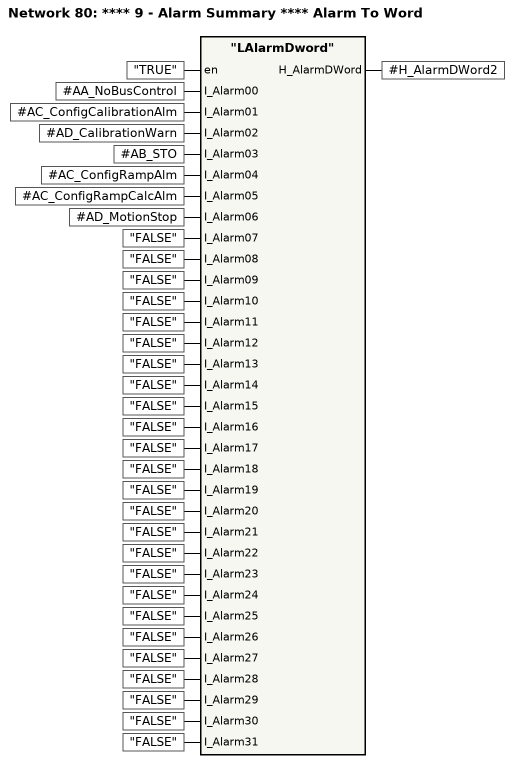
   IF "TRUE" THEN
       "LAlarmDword"(I_Alarm00 := #AA_NoBusControl,
                     I_Alarm01 := #AC_ConfigCalibrationAlm,
                     I_Alarm02 := #AD_CalibrationWarn,
                     I_Alarm03 := #AB_STO,
                     I_Alarm04 := #AC_ConfigRampAlm,
                     I_Alarm05 := #AC_ConfigRampCalcAlm,
                     I_Alarm06 := #AD_MotionStop,
                     I_Alarm07 := "FALSE",
                     I_Alarm08 := "FALSE",
                     I_Alarm09 := "FALSE",
                     I_Alarm10 := "FALSE",
                     I_Alarm11 := "FALSE",
                     I_Alarm12 := "FALSE",
                     I_Alarm13 := "FALSE",
                     I_Alarm14 := "FALSE",
                     I_Alarm15 := "FALSE",
                     I_Alarm16 := "FALSE",
                     I_Alarm17 := "FALSE",
                     I_Alarm18 := "FALSE",
                     I_Alarm19 := "FALSE",
                     I_Alarm20 := "FALSE",
                     I_Alarm21 := "FALSE",
                     I_Alarm22 := "FALSE",
                     I_Alarm23 := "FALSE",
                     I_Alarm24 := "FALSE",
                     I_Alarm25 := "FALSE",
                     I_Alarm26 := "FALSE",
                     I_Alarm27 := "FALSE",
                     I_Alarm28 := "FALSE",
                     I_Alarm29 := "FALSE",
                     I_Alarm30 := "FALSE",
                     I_Alarm31 := "FALSE",
                     H_AlarmDWord => #H_AlarmDWord2);
   END_IF;
END_REGION
END_FUNCTION_BLOCK
